LIN {X 0,Y 185.701,Z 460.549,A -85,B 0,C 180,E1 -22371.274,E2 -22371.274} C_VEL
LIN {X 0,Y 187.738,Z 470.881,A -85,B 0,C 180,E1 -22375.839,E2 -22375.839} C_VEL
LIN {X 0,Y 188.686,Z 475.361,A -85,B 0,C 180,E1 -22377.768,E2 -22377.768} C_VEL
LIN {X 0,Y 191.548,Z 486.797,A -85,B 0,C 180,E1 -22378.685,E2 -22378.685} C_VEL
LIN {X 0,Y 193.659,Z 519.979,A -85,B 0,C 180,E1 -22380.8,E2 -22380.8} C_VEL
LIN {X 0,Y 195.142,Z 539.248,A -85,B 0,C 180,E1 -22382.01,E2 -22382.01} C_VEL
LIN {X 0,Y 192.666,Z 586.047,A -85,B 0,C 180,E1 -22384.693,E2 -22384.693} C_VEL
LIN {X 0,Y 191.547,Z 599.858,A -85,B 0,C 180,E1 -22385.91,E2 -22385.91} C_VEL
LIN {X 0,Y 190.024,Z 613.54,A -85,B 0,C 180,E1 -22387.612,E2 -22387.612} C_VEL
LIN {X 0,Y 188.629,Z 625.455,A -85,B 0,C 180,E1 -22389.556,E2 -22389.556} C_VEL
LIN {X 0,Y 188.498,Z 626.394,A -85,B 0,C 180,E1 -22389.737,E2 -22389.737} C_VEL
LIN {X 0,Y 187.176,Z 631.288,A -85,B 0,C 180,E1 -22390.708,E2 -22390.708} C_VEL
LIN {X 0,Y 183.337,Z 638.645,A -85,B 0,C 180,E1 -22392.419,E2 -22392.419} C_VEL
LIN {X 0,Y 179.646,Z 645.469,A -85,B 0,C 180,E1 -22394.364,E2 -22394.364} C_VEL
LIN {X 0,Y 178.558,Z 649.547,A -85,B 0,C 180,E1 -22395.664,E2 -22395.664} C_VEL
LIN {X 0,Y 177.85,Z 657.711,A -85,B 0,C 180,E1 -22398.605,E2 -22398.605} C_VEL
LIN {X 0,Y 177.522,Z 664.858,A -85,B 0,C 180,E1 -22401.787,E2 -22401.787} C_VEL
LIN {X 0,Y 177.494,Z 671.375,A -85,B 0,C 180,E1 -22405.459,E2 -22405.459} C_VEL
LIN {X 0,Y 177.626,Z 675.992,A -85,B 0,C 180,E1 -22408.867,E2 -22408.867} C_VEL
LIN {X 0,Y 177.383,Z 678.317,A -85,B 0,C 180,E1 -22411.136,E2 -22411.136} C_VEL
LIN {X 0,Y 176.849,Z 680.76,A -85,B 0,C 180,E1 -22414.56,E2 -22414.56} C_VEL
LIN {X 0,Y 176.648,Z 681.882,A -85,B 0,C 180,E1 -22416.856,E2 -22416.856} C_VEL
LIN {X 0,Y 176.961,Z 682.934,A -85,B 0,C 180,E1 -22421.455,E2 -22421.455} C_VEL
LIN {X 0,Y 178.495,Z 682.536,A -85,B 0,C 180,E1 -22426,E2 -22426} C_VEL
LIN {X 0,Y 181.429,Z 680.73,A -85,B 0,C 180,E1 -22430.405,E2 -22430.405} C_VEL
LIN {X 0,Y 185.547,Z 677.444,A -85,B 0,C 180,E1 -22434.624,E2 -22434.624} C_VEL
LIN {X 0,Y 189.455,Z 673.992,A -85,B 0,C 180,E1 -22437.627,E2 -22437.627} C_VEL
LIN {X 0,Y 195.633,Z 667.93,A -85,B 0,C 180,E1 -22441.394,E2 -22441.394} C_VEL
LIN {X 0,Y 202.062,Z 661.103,A -85,B 0,C 180,E1 -22444.417,E2 -22444.417} C_VEL
LIN {X 0,Y 209.177,Z 652.611,A -85,B 0,C 180,E1 -22447.213,E2 -22447.213} C_VEL
LIN {X 0,Y 215.799,Z 643.753,A -85,B 0,C 180,E1 -22449.426,E2 -22449.426} C_VEL
LIN {X 0,Y 222.976,Z 632.961,A -85,B 0,C 180,E1 -22451.446,E2 -22451.446} C_VEL
LIN {X 0,Y 229.411,Z 621.99,A -85,B 0,C 180,E1 -22452.972,E2 -22452.972} C_VEL
LIN {X 0,Y 235.662,Z 609.39,A -85,B 0,C 180,E1 -22454.31,E2 -22454.31} C_VEL
LIN {X 0,Y 240.513,Z 597.54,A -85,B 0,C 180,E1 -22455.274,E2 -22455.274} C_VEL
LIN {X 0,Y 244.965,Z 584.543,A -85,B 0,C 180,E1 -22456.036,E2 -22456.036} C_VEL
LIN {X 0,Y 248.669,Z 569.68,A -85,B 0,C 180,E1 -22456.721,E2 -22456.721} C_VEL
LIN {X 0,Y 251.184,Z 556.435,A -85,B 0,C 180,E1 -22457.281,E2 -22457.281} C_VEL
LIN {X 0,Y 250.72,Z 552.705,A -85,B 0,C 180,E1 -22459.004,E2 -22459.004} C_VEL
LIN {X 0,Y 250.494,Z 550.56,A -85,B 0,C 180,E1 -22460.257,E2 -22460.257} C_VEL
LIN {X 0,Y 250.39,Z 547.96,A -85,B 0,C 180,E1 -22462.942,E2 -22462.942} C_VEL
LIN {X 0,Y 250.635,Z 547.364,A -85,B 0,C 180,E1 -22464.409,E2 -22464.409} C_VEL
LIN {X 0,Y 251.66,Z 547.678,A -85,B 0,C 180,E1 -22467.346,E2 -22467.346} C_VEL
LIN {X 0,Y 252.275,Z 548.822,A -85,B 0,C 180,E1 -22468.664,E2 -22468.664} C_VEL
LIN {X 0,Y 248.421,Z 568.129,A -85,B 0,C 180,E1 -22469.52,E2 -22469.52} C_VEL
LIN {X 0,Y 244.81,Z 581.444,A -85,B 0,C 180,E1 -22470.419,E2 -22470.419} C_VEL
LIN {X 0,Y 240.18,Z 594.192,A -85,B 0,C 180,E1 -22471.554,E2 -22471.554} C_VEL
LIN {X 0,Y 235.167,Z 605.631,A -85,B 0,C 180,E1 -22472.887,E2 -22472.887} C_VEL
LIN {X 0,Y 229.144,Z 616.854,A -85,B 0,C 180,E1 -22474.571,E2 -22474.571} C_VEL
LIN {X 0,Y 223.649,Z 625.549,A -85,B 0,C 180,E1 -22476.239,E2 -22476.239} C_VEL
LIN {X 0,Y 217.842,Z 633.74,A -85,B 0,C 180,E1 -22478.222,E2 -22478.222} C_VEL
LIN {X 0,Y 211.559,Z 641.305,A -85,B 0,C 180,E1 -22480.597,E2 -22480.597} C_VEL
LIN {X 0,Y 205.668,Z 647.446,A -85,B 0,C 180,E1 -22483.101,E2 -22483.101} C_VEL
LIN {X 0,Y 200.307,Z 652.348,A -85,B 0,C 180,E1 -22485.782,E2 -22485.782} C_VEL
LIN {X 0,Y 195.383,Z 656.121,A -85,B 0,C 180,E1 -22488.589,E2 -22488.589} C_VEL
LIN {X 0,Y 191.066,Z 658.891,A -85,B 0,C 180,E1 -22491.539,E2 -22491.539} C_VEL
LIN {X 0,Y 188.458,Z 660.203,A -85,B 0,C 180,E1 -22493.576,E2 -22493.576} C_VEL
LIN {X 0,Y 186.12,Z 661.109,A -85,B 0,C 180,E1 -22495.669,E2 -22495.669} C_VEL
LIN {X 0,Y 182.445,Z 661.688,A -85,B 0,C 180,E1 -22499.684,E2 -22499.684} C_VEL
LIN {X 0,Y 180.64,Z 661.354,A -85,B 0,C 180,E1 -22502.23,E2 -22502.23} C_VEL
LIN {X 0,Y 179.301,Z 660.645,A -85,B 0,C 180,E1 -22504.496,E2 -22504.496} C_VEL
LIN {X 0,Y 177.655,Z 658.413,A -85,B 0,C 180,E1 -22508.502,E2 -22508.502} C_VEL
LIN {X 0,Y 176.659,Z 654.746,A -85,B 0,C 180,E1 -22512.639,E2 -22512.639} C_VEL
LIN {X 0,Y 176.419,Z 650.464,A -85,B 0,C 180,E1 -22516.192,E2 -22516.192} C_VEL
LIN {X 0,Y 176.624,Z 643.895,A -85,B 0,C 180,E1 -22520.375,E2 -22520.375} C_VEL
LIN {X 0,Y 177.27,Z 636.508,A -85,B 0,C 180,E1 -22524.01,E2 -22524.01} C_VEL
LIN {X 0,Y 178.251,Z 627.333,A -85,B 0,C 180,E1 -22527.599,E2 -22527.599} C_VEL
LIN {X 0,Y 179.439,Z 617.727,A -85,B 0,C 180,E1 -22530.608,E2 -22530.608} C_VEL
LIN {X 0,Y 180.967,Z 605.843,A -85,B 0,C 180,E1 -22533.601,E2 -22533.601} C_VEL
LIN {X 0,Y 182.418,Z 593.758,A -85,B 0,C 180,E1 -22535.994,E2 -22535.994} C_VEL
LIN {X 0,Y 183.934,Z 580.594,A -85,B 0,C 180,E1 -22538.034,E2 -22538.034} C_VEL
LIN {X 0,Y 185.179,Z 566.664,A -85,B 0,C 180,E1 -22539.648,E2 -22539.648} C_VEL
LIN {X 0,Y 186.107,Z 553.364,A -85,B 0,C 180,E1 -22540.742,E2 -22540.742} C_VEL
LIN {X 0,Y 189.303,Z 493.801,A -85,B 0,C 180,E1 -22544.168,E2 -22544.168} C_VEL
LIN {X 0,Y 178.456,Z 461.253,A -85,B 0,C 180,E1 -22547.11,E2 -22547.11} C_VEL
LIN {X 0,Y 178.409,Z 461.26,A -85,B 0,C 180,E1 -22551.985,E2 -22551.985} C_VEL
LIN {X 0,Y 178.485,Z 461.252,A -85,B 0,C 180,E1 -22556.545,E2 -22556.545} C_VEL
LIN {X 0,Y 178.445,Z 461.254,A -85,B 0,C 180,E1 -22561.795,E2 -22561.795} C_VEL
LIN {X 0,Y 178.517,Z 461.247,A -85,B 0,C 180,E1 -22564.888,E2 -22564.888} C_VEL
LIN {X 0,Y 178.624,Z 461.23,A -85,B 0,C 180,E1 -22570.784,E2 -22570.784} C_VEL
LIN {X 0,Y 178.659,Z 461.232,A -85,B 0,C 180,E1 -22576.347,E2 -22576.347} C_VEL
LIN {X 0,Y 178.906,Z 461.196,A -85,B 0,C 180,E1 -22580.959,E2 -22580.959} C_VEL
LIN {X 0,Y 179.148,Z 461.166,A -85,B 0,C 180,E1 -22587.751,E2 -22587.751} C_VEL
LIN {X 0,Y 179.364,Z 461.138,A -85,B 0,C 180,E1 -22589.999,E2 -22589.999} C_VEL
LIN {X 0,Y 178.857,Z 461.206,A -85,B 0,C 180,E1 -22594.507,E2 -22594.507} C_VEL
LIN {X 0,Y 178.911,Z 461.196,A -85,B 0,C 180,E1 -22599.039,E2 -22599.039} C_VEL
LIN {X 0,Y 178.652,Z 461.229,A -85,B 0,C 180,E1 -22603.652,E2 -22603.652} C_VEL
LIN {X 0,Y 178.62,Z 461.234,A -85,B 0,C 180,E1 -22609.212,E2 -22609.212} C_VEL
LIN {X 0,Y 178.515,Z 461.243,A -85,B 0,C 180,E1 -22615.11,E2 -22615.11} C_VEL
LIN {X 0,Y 178.459,Z 461.255,A -85,B 0,C 180,E1 -22620.794,E2 -22620.794} C_VEL
LIN {X 0,Y 178.482,Z 461.248,A -85,B 0,C 180,E1 -22624.218,E2 -22624.218} C_VEL
LIN {X 0,Y 178.388,Z 461.263,A -85,B 0,C 180,E1 -22629.075,E2 -22629.075} C_VEL
LIN {X 0,Y 178.393,Z 461.26,A -85,B 0,C 180,E1 -22632.046,E2 -22632.046} C_VEL
LIN {X 0,Y 178.391,Z 461.262,A -85,B 0,C 180,E1 -22635.164,E2 -22635.164} C_VEL
LIN {X 0,Y 178.401,Z 461.263,A -85,B 0,C 180,E1 -22638.459,E2 -22638.459} C_VEL
LIN {X 0,Y 178.421,Z 461.257,A -85,B 0,C 180,E1 -22643.783,E2 -22643.783} C_VEL
LIN {X 0,Y 178.484,Z 461.254,A -85,B 0,C 180,E1 -22646.546,E2 -22646.546} C_VEL
LIN {X 0,Y 178.52,Z 461.243,A -85,B 0,C 180,E1 -22650.007,E2 -22650.007} C_VEL
LIN {X 0,Y 178.533,Z 461.246,A -85,B 0,C 180,E1 -22654.876,E2 -22654.876} C_VEL
LIN {X 0,Y 178.638,Z 461.232,A -85,B 0,C 180,E1 -22660.769,E2 -22660.769} C_VEL
LIN {X 0,Y 178.671,Z 461.228,A -85,B 0,C 180,E1 -22664.018,E2 -22664.018} C_VEL
LIN {X 0,Y 178.857,Z 461.203,A -85,B 0,C 180,E1 -22669.214,E2 -22669.214} C_VEL
LIN {X 0,Y 178.926,Z 461.195,A -85,B 0,C 180,E1 -22673.233,E2 -22673.233} C_VEL
LIN {X 0,Y 179.152,Z 461.165,A -85,B 0,C 180,E1 -22677.752,E2 -22677.752} C_VEL
LIN {X 0,Y 179.369,Z 461.141,A -85,B 0,C 180,E1 -22680,E2 -22680} C_VEL
LIN {X 0,Y 178.874,Z 461.2,A -85,B 0,C 180,E1 -22684.507,E2 -22684.507} C_VEL
LIN {X 0,Y 178.974,Z 461.191,A -85,B 0,C 180,E1 -22689.037,E2 -22689.037} C_VEL
LIN {X 0,Y 178.681,Z 461.221,A -85,B 0,C 180,E1 -22693.651,E2 -22693.651} C_VEL
LIN {X 0,Y 178.621,Z 461.234,A -85,B 0,C 180,E1 -22699.216,E2 -22699.216} C_VEL
LIN {X 0,Y 178.519,Z 461.247,A -85,B 0,C 180,E1 -22705.115,E2 -22705.115} C_VEL
LIN {X 0,Y 178.501,Z 461.246,A -85,B 0,C 180,E1 -22710.787,E2 -22710.787} C_VEL
LIN {X 0,Y 178.485,Z 461.251,A -85,B 0,C 180,E1 -22714.22,E2 -22714.22} C_VEL
LIN {X 0,Y 178.395,Z 461.258,A -85,B 0,C 180,E1 -22719.075,E2 -22719.075} C_VEL
LIN {X 0,Y 178.398,Z 461.26,A -85,B 0,C 180,E1 -22722.045,E2 -22722.045} C_VEL
LIN {X 0,Y 178.394,Z 461.263,A -85,B 0,C 180,E1 -22725.164,E2 -22725.164} C_VEL
LIN {X 0,Y 178.599,Z 461.379,A -85,B 0,C 180,E1 -22730.979,E2 -22730.979} C_VEL
LIN {X 0,Y 180.643,Z 471.556,A -85,B 0,C 180,E1 -22735.659,E2 -22735.659} C_VEL
LIN {X 0,Y 181.369,Z 475.028,A -85,B 0,C 180,E1 -22737.147,E2 -22737.147} C_VEL
LIN {X 0,Y 184.69,Z 487.892,A -85,B 0,C 180,E1 -22738.233,E2 -22738.233} C_VEL
LIN {X 0,Y 186.699,Z 520.317,A -85,B 0,C 180,E1 -22740.381,E2 -22740.381} C_VEL
LIN {X 0,Y 188.159,Z 539.471,A -85,B 0,C 180,E1 -22741.637,E2 -22741.637} C_VEL
LIN {X 0,Y 185.629,Z 585.844,A -85,B 0,C 180,E1 -22744.416,E2 -22744.416} C_VEL
LIN {X 0,Y 184.49,Z 599.914,A -85,B 0,C 180,E1 -22745.722,E2 -22745.722} C_VEL
LIN {X 0,Y 182.927,Z 613.572,A -85,B 0,C 180,E1 -22747.508,E2 -22747.508} C_VEL
LIN {X 0,Y 181.442,Z 625.783,A -85,B 0,C 180,E1 -22749.616,E2 -22749.616} C_VEL
LIN {X 0,Y 180.084,Z 637.05,A -85,B 0,C 180,E1 -22752.102,E2 -22752.102} C_VEL
LIN {X 0,Y 178.904,Z 646.257,A -85,B 0,C 180,E1 -22754.624,E2 -22754.624} C_VEL
LIN {X 0,Y 178.558,Z 649.547,A -85,B 0,C 180,E1 -22755.664,E2 -22755.664} C_VEL
LIN {X 0,Y 177.546,Z 653.521,A -85,B 0,C 180,E1 -22757.032,E2 -22757.032} C_VEL
LIN {X 0,Y 174.285,Z 659.229,A -85,B 0,C 180,E1 -22759.452,E2 -22759.452} C_VEL
LIN {X 0,Y 171.212,Z 664.277,A -85,B 0,C 180,E1 -22762.125,E2 -22762.125} C_VEL
LIN {X 0,Y 170.513,Z 667.229,A -85,B 0,C 180,E1 -22763.845,E2 -22763.845} C_VEL
LIN {X 0,Y 170.596,Z 672.954,A -85,B 0,C 180,E1 -22767.64,E2 -22767.64} C_VEL
LIN {X 0,Y 170.668,Z 675.747,A -85,B 0,C 180,E1 -22770.001,E2 -22770.001} C_VEL
LIN {X 0,Y 170.245,Z 677.883,A -85,B 0,C 180,E1 -22772.367,E2 -22772.367} C_VEL
LIN {X 0,Y 169.72,Z 680.438,A -85,B 0,C 180,E1 -22776.368,E2 -22776.368} C_VEL
LIN {X 0,Y 169.645,Z 681.621,A -85,B 0,C 180,E1 -22779.539,E2 -22779.539} C_VEL
LIN {X 0,Y 170.666,Z 682.248,A -85,B 0,C 180,E1 -22784.306,E2 -22784.306} C_VEL
LIN {X 0,Y 173.115,Z 681.425,A -85,B 0,C 180,E1 -22788.953,E2 -22788.953} C_VEL
LIN {X 0,Y 176.794,Z 679.2,A -85,B 0,C 180,E1 -22793.425,E2 -22793.425} C_VEL
LIN {X 0,Y 181.757,Z 675.549,A -85,B 0,C 180,E1 -22797.647,E2 -22797.647} C_VEL
LIN {X 0,Y 186.362,Z 671.786,A -85,B 0,C 180,E1 -22800.605,E2 -22800.605} C_VEL
LIN {X 0,Y 191.512,Z 667.071,A -85,B 0,C 180,E1 -22803.4,E2 -22803.4} C_VEL
LIN {X 0,Y 198.38,Z 660.316,A -85,B 0,C 180,E1 -22806.4,E2 -22806.4} C_VEL
LIN {X 0,Y 204.815,Z 653.196,A -85,B 0,C 180,E1 -22808.773,E2 -22808.773} C_VEL
LIN {X 0,Y 211.719,Z 644.664,A -85,B 0,C 180,E1 -22810.966,E2 -22810.966} C_VEL
LIN {X 0,Y 219.17,Z 634.332,A -85,B 0,C 180,E1 -22812.955,E2 -22812.955} C_VEL
LIN {X 0,Y 225.823,Z 623.791,A -85,B 0,C 180,E1 -22814.447,E2 -22814.447} C_VEL
LIN {X 0,Y 231.994,Z 612.482,A -85,B 0,C 180,E1 -22815.7,E2 -22815.7} C_VEL
LIN {X 0,Y 237.79,Z 599.752,A -85,B 0,C 180,E1 -22816.782,E2 -22816.782} C_VEL
LIN {X 0,Y 242.47,Z 587.137,A -85,B 0,C 180,E1 -22817.529,E2 -22817.529} C_VEL
LIN {X 0,Y 246.909,Z 571.217,A -85,B 0,C 180,E1 -22818.276,E2 -22818.276} C_VEL
LIN {X 0,Y 249.076,Z 560.769,A -85,B 0,C 180,E1 -22818.712,E2 -22818.712} C_VEL
LIN {X 0,Y 248.802,Z 557.233,A -85,B 0,C 180,E1 -22820.64,E2 -22820.64} C_VEL
LIN {X 0,Y 248.861,Z 554.658,A -85,B 0,C 180,E1 -22823.383,E2 -22823.383} C_VEL
LIN {X 0,Y 249.34,Z 554.291,A -85,B 0,C 180,E1 -22825.686,E2 -22825.686} C_VEL
LIN {X 0,Y 250.017,Z 554.637,A -85,B 0,C 180,E1 -22827.235,E2 -22827.235} C_VEL
LIN {X 0,Y 246.333,Z 571.491,A -85,B 0,C 180,E1 -22828.075,E2 -22828.075} C_VEL
LIN {X 0,Y 242.221,Z 584.894,A -85,B 0,C 180,E1 -22829.001,E2 -22829.001} C_VEL
LIN {X 0,Y 237.736,Z 596.488,A -85,B 0,C 180,E1 -22830.057,E2 -22830.057} C_VEL
LIN {X 0,Y 232.572,Z 607.309,A -85,B 0,C 180,E1 -22831.319,E2 -22831.319} C_VEL
LIN {X 0,Y 225.615,Z 619.36,A -85,B 0,C 180,E1 -22833.148,E2 -22833.148} C_VEL
LIN {X 0,Y 219.543,Z 628.275,A -85,B 0,C 180,E1 -22834.902,E2 -22834.902} C_VEL
LIN {X 0,Y 212.619,Z 636.953,A -85,B 0,C 180,E1 -22837.145,E2 -22837.145} C_VEL
LIN {X 0,Y 206.117,Z 644.087,A -85,B 0,C 180,E1 -22839.543,E2 -22839.543} C_VEL
LIN {X 0,Y 200.931,Z 648.956,A -85,B 0,C 180,E1 -22841.651,E2 -22841.651} C_VEL
LIN {X 0,Y 195.276,Z 653.63,A -85,B 0,C 180,E1 -22844.34,E2 -22844.34} C_VEL
LIN {X 0,Y 190.04,Z 657.289,A -85,B 0,C 180,E1 -22847.18,E2 -22847.18} C_VEL
LIN {X 0,Y 185.499,Z 659.837,A -85,B 0,C 180,E1 -22850.09,E2 -22850.09} C_VEL
LIN {X 0,Y 181.3,Z 661.572,A -85,B 0,C 180,E1 -22853.322,E2 -22853.322} C_VEL
LIN {X 0,Y 176.771,Z 662.426,A -85,B 0,C 180,E1 -22857.721,E2 -22857.721} C_VEL
LIN {X 0,Y 174.956,Z 662.226,A -85,B 0,C 180,E1 -22860,E2 -22860} C_VEL
LIN {X 0,Y 172.03,Z 660.637,A -85,B 0,C 180,E1 -22864.687,E2 -22864.687} C_VEL
LIN {X 0,Y 170.54,Z 658.221,A -85,B 0,C 180,E1 -22868.481,E2 -22868.481} C_VEL
LIN {X 0,Y 169.664,Z 655.105,A -85,B 0,C 180,E1 -22871.953,E2 -22871.953} C_VEL
LIN {X 0,Y 169.34,Z 650.753,A -85,B 0,C 180,E1 -22875.65,E2 -22875.65} C_VEL
LIN {X 0,Y 169.442,Z 645.131,A -85,B 0,C 180,E1 -22879.379,E2 -22879.379} C_VEL
LIN {X 0,Y 169.988,Z 638.049,A -85,B 0,C 180,E1 -22883.127,E2 -22883.127} C_VEL
LIN {X 0,Y 170.962,Z 629.103,A -85,B 0,C 180,E1 -22886.884,E2 -22886.884} C_VEL
LIN {X 0,Y 172.01,Z 620.202,A -85,B 0,C 180,E1 -22889.922,E2 -22889.922} C_VEL
LIN {X 0,Y 173.341,Z 609.586,A -85,B 0,C 180,E1 -22892.839,E2 -22892.839} C_VEL
LIN {X 0,Y 174.77,Z 598.414,A -85,B 0,C 180,E1 -22895.314,E2 -22895.314} C_VEL
LIN {X 0,Y 176.285,Z 586.092,A -85,B 0,C 180,E1 -22897.484,E2 -22897.484} C_VEL
LIN {X 0,Y 177.597,Z 572.798,A -85,B 0,C 180,E1 -22899.284,E2 -22899.284} C_VEL
LIN {X 0,Y 178.742,Z 559.118,A -85,B 0,C 180,E1 -22900.634,E2 -22900.634} C_VEL
LIN {X 0,Y 179.933,Z 536.769,A -85,B 0,C 180,E1 -22902.096,E2 -22902.096} C_VEL
LIN {X 0,Y 182.328,Z 494.869,A -85,B 0,C 180,E1 -22904.608,E2 -22904.608} C_VEL
LIN {X 0,Y 171.384,Z 462.134,A -85,B 0,C 180,E1 -22907.705,E2 -22907.705} C_VEL
LIN {X 0,Y 171.361,Z 462.139,A -85,B 0,C 180,E1 -22912.033,E2 -22912.033} C_VEL
LIN {X 0,Y 171.399,Z 462.131,A -85,B 0,C 180,E1 -22915.092,E2 -22915.092} C_VEL
LIN {X 0,Y 171.41,Z 462.132,A -85,B 0,C 180,E1 -22920.526,E2 -22920.526} C_VEL
LIN {X 0,Y 171.444,Z 462.127,A -85,B 0,C 180,E1 -22925.799,E2 -22925.799} C_VEL
LIN {X 0,Y 171.58,Z 462.106,A -85,B 0,C 180,E1 -22930.871,E2 -22930.871} C_VEL
LIN {X 0,Y 171.577,Z 462.112,A -85,B 0,C 180,E1 -22935.772,E2 -22935.772} C_VEL
LIN {X 0,Y 171.844,Z 462.075,A -85,B 0,C 180,E1 -22940.584,E2 -22940.584} C_VEL
LIN {X 0,Y 171.804,Z 462.083,A -85,B 0,C 180,E1 -22945.306,E2 -22945.306} C_VEL
LIN {X 0,Y 172.328,Z 462.014,A -85,B 0,C 180,E1 -22949.999,E2 -22949.999} C_VEL
LIN {X 0,Y 171.806,Z 462.083,A -85,B 0,C 180,E1 -22954.692,E2 -22954.692} C_VEL
LIN {X 0,Y 171.848,Z 462.075,A -85,B 0,C 180,E1 -22959.414,E2 -22959.414} C_VEL
LIN {X 0,Y 171.569,Z 462.113,A -85,B 0,C 180,E1 -22964.227,E2 -22964.227} C_VEL
LIN {X 0,Y 171.539,Z 462.115,A -85,B 0,C 180,E1 -22969.555,E2 -22969.555} C_VEL
LIN {X 0,Y 171.443,Z 462.123,A -85,B 0,C 180,E1 -22975.598,E2 -22975.598} C_VEL
LIN {X 0,Y 171.417,Z 462.133,A -85,B 0,C 180,E1 -22980.572,E2 -22980.572} C_VEL
LIN {X 0,Y 171.391,Z 462.133,A -85,B 0,C 180,E1 -22985.034,E2 -22985.034} C_VEL
LIN {X 0,Y 171.343,Z 462.142,A -85,B 0,C 180,E1 -22988.801,E2 -22988.801} C_VEL
LIN {X 0,Y 171.318,Z 462.141,A -85,B 0,C 180,E1 -22994.217,E2 -22994.217} C_VEL
LIN {X 0,Y 171.334,Z 462.141,A -85,B 0,C 180,E1 -22998.981,E2 -22998.981} C_VEL
LIN {X 0,Y 171.385,Z 462.13,A -85,B 0,C 180,E1 -23002.041,E2 -23002.041} C_VEL
LIN {X 0,Y 171.397,Z 462.135,A -85,B 0,C 180,E1 -23005.092,E2 -23005.092} C_VEL
LIN {X 0,Y 171.447,Z 462.124,A -85,B 0,C 180,E1 -23010.534,E2 -23010.534} C_VEL
LIN {X 0,Y 171.458,Z 462.126,A -85,B 0,C 180,E1 -23015.802,E2 -23015.802} C_VEL
LIN {X 0,Y 171.594,Z 462.11,A -85,B 0,C 180,E1 -23020.874,E2 -23020.874} C_VEL
LIN {X 0,Y 171.596,Z 462.107,A -85,B 0,C 180,E1 -23025.775,E2 -23025.775} C_VEL
LIN {X 0,Y 171.889,Z 462.074,A -85,B 0,C 180,E1 -23030.587,E2 -23030.587} C_VEL
LIN {X 0,Y 171.82,Z 462.077,A -85,B 0,C 180,E1 -23035.308,E2 -23035.308} C_VEL
LIN {X 0,Y 172.332,Z 462.017,A -85,B 0,C 180,E1 -23040,E2 -23040} C_VEL
LIN {X 0,Y 171.823,Z 462.078,A -85,B 0,C 180,E1 -23044.693,E2 -23044.693} C_VEL
LIN {X 0,Y 171.907,Z 462.07,A -85,B 0,C 180,E1 -23049.412,E2 -23049.412} C_VEL
LIN {X 0,Y 171.594,Z 462.105,A -85,B 0,C 180,E1 -23054.226,E2 -23054.226} C_VEL
LIN {X 0,Y 171.541,Z 462.115,A -85,B 0,C 180,E1 -23059.56,E2 -23059.56} C_VEL
LIN {X 0,Y 171.458,Z 462.126,A -85,B 0,C 180,E1 -23065.61,E2 -23065.61} C_VEL
LIN {X 0,Y 171.458,Z 462.124,A -85,B 0,C 180,E1 -23070.597,E2 -23070.597} C_VEL
LIN {X 0,Y 171.392,Z 462.136,A -85,B 0,C 180,E1 -23075.035,E2 -23075.035} C_VEL
LIN {X 0,Y 171.357,Z 462.136,A -85,B 0,C 180,E1 -23078.808,E2 -23078.808} C_VEL
LIN {X 0,Y 171.321,Z 462.144,A -85,B 0,C 180,E1 -23084.218,E2 -23084.218} C_VEL
LIN {X 0,Y 171.502,Z 462.119,A -85,B 0,C 180,E1 -23090.579,E2 -23090.579} C_VEL
LIN {X 0,Y 173.542,Z 472.168,A -85,B 0,C 180,E1 -23095.462,E2 -23095.462} C_VEL
LIN {X 0,Y 173.972,Z 474.305,A -85,B 0,C 180,E1 -23096.459,E2 -23096.459} C_VEL
LIN {X 0,Y 177.844,Z 489.066,A -85,B 0,C 180,E1 -23097.756,E2 -23097.756} C_VEL
LIN {X 0,Y 179.756,Z 520.758,A -85,B 0,C 180,E1 -23099.937,E2 -23099.937} C_VEL
LIN {X 0,Y 181.179,Z 540.044,A -85,B 0,C 180,E1 -23101.264,E2 -23101.264} C_VEL
LIN {X 0,Y 178.679,Z 584.578,A -85,B 0,C 180,E1 -23104.051,E2 -23104.051} C_VEL
LIN {X 0,Y 177.556,Z 598.633,A -85,B 0,C 180,E1 -23105.396,E2 -23105.396} C_VEL
LIN {X 0,Y 175.989,Z 611.81,A -85,B 0,C 180,E1 -23107.165,E2 -23107.165} C_VEL
LIN {X 0,Y 174.49,Z 624.286,A -85,B 0,C 180,E1 -23109.365,E2 -23109.365} C_VEL
LIN {X 0,Y 173.118,Z 635.756,A -85,B 0,C 180,E1 -23111.969,E2 -23111.969} C_VEL
LIN {X 0,Y 171.904,Z 645.068,A -85,B 0,C 180,E1 -23114.59,E2 -23114.59} C_VEL
LIN {X 0,Y 171.148,Z 653.703,A -85,B 0,C 180,E1 -23117.551,E2 -23117.551} C_VEL
LIN {X 0,Y 170.577,Z 661.794,A -85,B 0,C 180,E1 -23121.012,E2 -23121.012} C_VEL
LIN {X 0,Y 170.513,Z 667.229,A -85,B 0,C 180,E1 -23123.845,E2 -23123.845} C_VEL
LIN {X 0,Y 169.84,Z 669.942,A -85,B 0,C 180,E1 -23125.605,E2 -23125.605} C_VEL
LIN {X 0,Y 168.256,Z 672.115,A -85,B 0,C 180,E1 -23127.404,E2 -23127.404} C_VEL
LIN {X 0,Y 164.424,Z 675.542,A -85,B 0,C 180,E1 -23131.183,E2 -23131.183} C_VEL
LIN {X 0,Y 163.025,Z 677.475,A -85,B 0,C 180,E1 -23133.88,E2 -23133.88} C_VEL
LIN {X 0,Y 162.658,Z 679.622,A -85,B 0,C 180,E1 -23137.449,E2 -23137.449} C_VEL
LIN {X 0,Y 163.067,Z 681.206,A -85,B 0,C 180,E1 -23142.445,E2 -23142.445} C_VEL
LIN {X 0,Y 164.867,Z 681.393,A -85,B 0,C 180,E1 -23147.362,E2 -23147.362} C_VEL
LIN {X 0,Y 168.164,Z 680.215,A -85,B 0,C 180,E1 -23152.095,E2 -23152.095} C_VEL
LIN {X 0,Y 172.733,Z 677.628,A -85,B 0,C 180,E1 -23156.588,E2 -23156.588} C_VEL
LIN {X 0,Y 178.616,Z 673.581,A -85,B 0,C 180,E1 -23160.765,E2 -23160.765} C_VEL
LIN {X 0,Y 185.676,Z 668.028,A -85,B 0,C 180,E1 -23164.596,E2 -23164.596} C_VEL
LIN {X 0,Y 192.807,Z 661.677,A -85,B 0,C 180,E1 -23167.631,E2 -23167.631} C_VEL
LIN {X 0,Y 200.613,Z 653.822,A -85,B 0,C 180,E1 -23170.4,E2 -23170.4} C_VEL
LIN {X 0,Y 207.8,Z 645.644,A -85,B 0,C 180,E1 -23172.566,E2 -23172.566} C_VEL
LIN {X 0,Y 215.529,Z 635.756,A -85,B 0,C 180,E1 -23174.514,E2 -23174.514} C_VEL
LIN {X 0,Y 221.831,Z 626.654,A -85,B 0,C 180,E1 -23175.858,E2 -23175.858} C_VEL
LIN {X 0,Y 228.713,Z 615.037,A -85,B 0,C 180,E1 -23177.193,E2 -23177.193} C_VEL
LIN {X 0,Y 235.227,Z 601.98,A -85,B 0,C 180,E1 -23178.327,E2 -23178.327} C_VEL
LIN {X 0,Y 240.808,Z 588.272,A -85,B 0,C 180,E1 -23179.137,E2 -23179.137} C_VEL
LIN {X 0,Y 245.118,Z 574.249,A -85,B 0,C 180,E1 -23179.793,E2 -23179.793} C_VEL
LIN {X 0,Y 247.164,Z 565.427,A -85,B 0,C 180,E1 -23180.196,E2 -23180.196} C_VEL
LIN {X 0,Y 247.177,Z 563.443,A -85,B 0,C 180,E1 -23181.454,E2 -23181.454} C_VEL
LIN {X 0,Y 247.349,Z 561.484,A -85,B 0,C 180,E1 -23183.677,E2 -23183.677} C_VEL
LIN {X 0,Y 247.841,Z 561.257,A -85,B 0,C 180,E1 -23185.916,E2 -23185.916} C_VEL
LIN {X 0,Y 245.069,Z 572.959,A -85,B 0,C 180,E1 -23186.487,E2 -23186.487} C_VEL
LIN {X 0,Y 240.86,Z 585.994,A -85,B 0,C 180,E1 -23187.366,E2 -23187.366} C_VEL
LIN {X 0,Y 236.172,Z 597.354,A -85,B 0,C 180,E1 -23188.366,E2 -23188.366} C_VEL
LIN {X 0,Y 229.451,Z 610.476,A -85,B 0,C 180,E1 -23189.911,E2 -23189.911} C_VEL
LIN {X 0,Y 222.995,Z 620.916,A -85,B 0,C 180,E1 -23191.505,E2 -23191.505} C_VEL
LIN {X 0,Y 215.897,Z 630.475,A -85,B 0,C 180,E1 -23193.41,E2 -23193.41} C_VEL
LIN {X 0,Y 209.725,Z 637.799,A -85,B 0,C 180,E1 -23195.3,E2 -23195.3} C_VEL
LIN {X 0,Y 202.938,Z 644.733,A -85,B 0,C 180,E1 -23197.608,E2 -23197.608} C_VEL
LIN {X 0,Y 196.367,Z 650.493,A -85,B 0,C 180,E1 -23200.122,E2 -23200.122} C_VEL
LIN {X 0,Y 190.387,Z 655.006,A -85,B 0,C 180,E1 -23202.823,E2 -23202.823} C_VEL
LIN {X 0,Y 183.084,Z 659.375,A -85,B 0,C 180,E1 -23206.684,E2 -23206.684} C_VEL
LIN {X 0,Y 178.664,Z 661.412,A -85,B 0,C 180,E1 -23209.555,E2 -23209.555} C_VEL
LIN {X 0,Y 174.137,Z 662.773,A -85,B 0,C 180,E1 -23213.046,E2 -23213.046} C_VEL
LIN {X 0,Y 169.515,Z 663.047,A -85,B 0,C 180,E1 -23217.624,E2 -23217.624} C_VEL
LIN {X 0,Y 167.69,Z 662.597,A -85,B 0,C 180,E1 -23220,E2 -23220} C_VEL
LIN {X 0,Y 164.745,Z 660.451,A -85,B 0,C 180,E1 -23224.894,E2 -23224.894} C_VEL
LIN {X 0,Y 163.428,Z 657.93,A -85,B 0,C 180,E1 -23228.466,E2 -23228.466} C_VEL
LIN {X 0,Y 162.503,Z 654.056,A -85,B 0,C 180,E1 -23232.488,E2 -23232.488} C_VEL
LIN {X 0,Y 162.235,Z 649.229,A -85,B 0,C 180,E1 -23236.354,E2 -23236.354} C_VEL
LIN {X 0,Y 162.461,Z 643.09,A -85,B 0,C 180,E1 -23240.247,E2 -23240.247} C_VEL
LIN {X 0,Y 163.143,Z 635.348,A -85,B 0,C 180,E1 -23244.158,E2 -23244.158} C_VEL
LIN {X 0,Y 164.016,Z 627.333,A -85,B 0,C 180,E1 -23247.428,E2 -23247.428} C_VEL
LIN {X 0,Y 165.218,Z 617.558,A -85,B 0,C 180,E1 -23250.694,E2 -23250.694} C_VEL
LIN {X 0,Y 166.635,Z 606.81,A -85,B 0,C 180,E1 -23253.611,E2 -23253.611} C_VEL
LIN {X 0,Y 168.106,Z 594.952,A -85,B 0,C 180,E1 -23256.175,E2 -23256.175} C_VEL
LIN {X 0,Y 169.517,Z 583.239,A -85,B 0,C 180,E1 -23258.185,E2 -23258.185} C_VEL
LIN {X 0,Y 170.774,Z 570.774,A -85,B 0,C 180,E1 -23259.826,E2 -23259.826} C_VEL
LIN {X 0,Y 171.936,Z 556.02,A -85,B 0,C 180,E1 -23261.233,E2 -23261.233} C_VEL
LIN {X 0,Y 175.274,Z 495.88,A -85,B 0,C 180,E1 -23265.056,E2 -23265.056} C_VEL
LIN {X 0,Y 164.331,Z 463.015,A -85,B 0,C 180,E1 -23268.324,E2 -23268.324} C_VEL
LIN {X 0,Y 164.327,Z 463.011,A -85,B 0,C 180,E1 -23274.351,E2 -23274.351} C_VEL
LIN {X 0,Y 164.372,Z 463.009,A -85,B 0,C 180,E1 -23279.13,E2 -23279.13} C_VEL
LIN {X 0,Y 164.397,Z 463.006,A -85,B 0,C 180,E1 -23284.69,E2 -23284.69} C_VEL
LIN {X 0,Y 164.486,Z 462.994,A -85,B 0,C 180,E1 -23290.051,E2 -23290.051} C_VEL
LIN {X 0,Y 164.525,Z 462.99,A -85,B 0,C 180,E1 -23295.148,E2 -23295.148} C_VEL
LIN {X 0,Y 164.766,Z 462.956,A -85,B 0,C 180,E1 -23300.175,E2 -23300.175} C_VEL
LIN {X 0,Y 164.823,Z 462.954,A -85,B 0,C 180,E1 -23302.65,E2 -23302.65} C_VEL
LIN {X 0,Y 165.043,Z 462.923,A -85,B 0,C 180,E1 -23307.559,E2 -23307.559} C_VEL
LIN {X 0,Y 165.291,Z 462.89,A -85,B 0,C 180,E1 -23309.999,E2 -23309.999} C_VEL
LIN {X 0,Y 164.755,Z 462.961,A -85,B 0,C 180,E1 -23314.893,E2 -23314.893} C_VEL
LIN {X 0,Y 164.828,Z 462.947,A -85,B 0,C 180,E1 -23317.348,E2 -23317.348} C_VEL
LIN {X 0,Y 164.703,Z 462.968,A -85,B 0,C 180,E1 -23321.06,E2 -23321.06} C_VEL
LIN {X 0,Y 164.477,Z 462.992,A -85,B 0,C 180,E1 -23327.403,E2 -23327.403} C_VEL
LIN {X 0,Y 164.472,Z 462.996,A -85,B 0,C 180,E1 -23329.988,E2 -23329.988} C_VEL
LIN {X 0,Y 164.37,Z 463.005,A -85,B 0,C 180,E1 -23336.116,E2 -23336.116} C_VEL
LIN {X 0,Y 164.357,Z 463.01,A -85,B 0,C 180,E1 -23341.217,E2 -23341.217} C_VEL
LIN {X 0,Y 164.279,Z 463.022,A -85,B 0,C 180,E1 -23346.792,E2 -23346.792} C_VEL
LIN {X 0,Y 164.285,Z 463.02,A -85,B 0,C 180,E1 -23349.917,E2 -23349.917} C_VEL
LIN {X 0,Y 164.278,Z 463.017,A -85,B 0,C 180,E1 -23353.341,E2 -23353.341} C_VEL
LIN {X 0,Y 164.262,Z 463.024,A -85,B 0,C 180,E1 -23356.799,E2 -23356.799} C_VEL
LIN {X 0,Y 164.294,Z 463.017,A -85,B 0,C 180,E1 -23360.351,E2 -23360.351} C_VEL
LIN {X 0,Y 164.329,Z 463.014,A -85,B 0,C 180,E1 -23364.349,E2 -23364.349} C_VEL
LIN {X 0,Y 164.388,Z 463.003,A -85,B 0,C 180,E1 -23369.134,E2 -23369.134} C_VEL
LIN {X 0,Y 164.415,Z 463.006,A -85,B 0,C 180,E1 -23374.694,E2 -23374.694} C_VEL
LIN {X 0,Y 164.485,Z 462.991,A -85,B 0,C 180,E1 -23380.05,E2 -23380.05} C_VEL
LIN {X 0,Y 164.547,Z 462.986,A -85,B 0,C 180,E1 -23385.151,E2 -23385.151} C_VEL
LIN {X 0,Y 164.803,Z 462.954,A -85,B 0,C 180,E1 -23390.179,E2 -23390.179} C_VEL
LIN {X 0,Y 164.852,Z 462.951,A -85,B 0,C 180,E1 -23392.652,E2 -23392.652} C_VEL
LIN {X 0,Y 165.048,Z 462.922,A -85,B 0,C 180,E1 -23397.56,E2 -23397.56} C_VEL
LIN {X 0,Y 165.295,Z 462.894,A -85,B 0,C 180,E1 -23400,E2 -23400} C_VEL
LIN {X 0,Y 164.773,Z 462.955,A -85,B 0,C 180,E1 -23404.894,E2 -23404.894} C_VEL
LIN {X 0,Y 164.85,Z 462.949,A -85,B 0,C 180,E1 -23409.819,E2 -23409.819} C_VEL
LIN {X 0,Y 164.536,Z 462.986,A -85,B 0,C 180,E1 -23414.85,E2 -23414.85} C_VEL
LIN {X 0,Y 164.472,Z 462.996,A -85,B 0,C 180,E1 -23419.99,E2 -23419.99} C_VEL
LIN {X 0,Y 164.385,Z 463.007,A -85,B 0,C 180,E1 -23426.129,E2 -23426.129} C_VEL
LIN {X 0,Y 164.388,Z 463.003,A -85,B 0,C 180,E1 -23431.236,E2 -23431.236} C_VEL
LIN {X 0,Y 164.294,Z 463.02,A -85,B 0,C 180,E1 -23436.79,E2 -23436.79} C_VEL
LIN {X 0,Y 164.29,Z 463.014,A -85,B 0,C 180,E1 -23439.917,E2 -23439.917} C_VEL
LIN {X 0,Y 164.279,Z 463.021,A -85,B 0,C 180,E1 -23443.343,E2 -23443.343} C_VEL
LIN {X 0,Y 164.292,Z 463.018,A -85,B 0,C 180,E1 -23446.809,E2 -23446.809} C_VEL
LIN {X 0,Y 164.482,Z 463.193,A -85,B 0,C 180,E1 -23450.514,E2 -23450.514} C_VEL
LIN {X 0,Y 166.49,Z 473.019,A -85,B 0,C 180,E1 -23455.402,E2 -23455.402} C_VEL
LIN {X 0,Y 166.654,Z 473.881,A -85,B 0,C 180,E1 -23455.774,E2 -23455.774} C_VEL
LIN {X 0,Y 170.974,Z 491.005,A -85,B 0,C 180,E1 -23457.338,E2 -23457.338} C_VEL
LIN {X 0,Y 173.094,Z 525.175,A -85,B 0,C 180,E1 -23459.811,E2 -23459.811} C_VEL
LIN {X 0,Y 174.205,Z 540.086,A -85,B 0,C 180,E1 -23460.874,E2 -23460.874} C_VEL
LIN {X 0,Y 171.598,Z 585.066,A -85,B 0,C 180,E1 -23463.855,E2 -23463.855} C_VEL
LIN {X 0,Y 170.511,Z 598.152,A -85,B 0,C 180,E1 -23465.177,E2 -23465.177} C_VEL
LIN {X 0,Y 169.049,Z 610.362,A -85,B 0,C 180,E1 -23466.867,E2 -23466.867} C_VEL
LIN {X 0,Y 167.554,Z 622.8,A -85,B 0,C 180,E1 -23469.114,E2 -23469.114} C_VEL
LIN {X 0,Y 166.125,Z 634.446,A -85,B 0,C 180,E1 -23471.821,E2 -23471.821} C_VEL
LIN {X 0,Y 164.918,Z 643.884,A -85,B 0,C 180,E1 -23474.554,E2 -23474.554} C_VEL
LIN {X 0,Y 164.136,Z 652.603,A -85,B 0,C 180,E1 -23477.639,E2 -23477.639} C_VEL
LIN {X 0,Y 163.611,Z 660.469,A -85,B 0,C 180,E1 -23481.108,E2 -23481.108} C_VEL
LIN {X 0,Y 163.566,Z 666.617,A -85,B 0,C 180,E1 -23484.453,E2 -23484.453} C_VEL
LIN {X 0,Y 163.636,Z 671.207,A -85,B 0,C 180,E1 -23487.539,E2 -23487.539} C_VEL
LIN {X 0,Y 163.737,Z 674.15,A -85,B 0,C 180,E1 -23490.001,E2 -23490.001} C_VEL
LIN {X 0,Y 163.025,Z 677.475,A -85,B 0,C 180,E1 -23493.88,E2 -23493.88} C_VEL
LIN {X 0,Y 162.122,Z 678.693,A -85,B 0,C 180,E1 -23495.889,E2 -23495.889} C_VEL
LIN {X 0,Y 159.191,Z 679.759,A -85,B 0,C 180,E1 -23499.244,E2 -23499.244} C_VEL
LIN {X 0,Y 157.084,Z 680.183,A -85,B 0,C 180,E1 -23502.032,E2 -23502.032} C_VEL
LIN {X 0,Y 156.551,Z 680.474,A -85,B 0,C 180,E1 -23504.192,E2 -23504.192} C_VEL
LIN {X 0,Y 156.693,Z 680.55,A -85,B 0,C 180,E1 -23504.913,E2 -23504.913} C_VEL
LIN {X 0,Y 158.1,Z 680.737,A -85,B 0,C 180,E1 -23508.131,E2 -23508.131} C_VEL
LIN {X 0,Y 161.596,Z 679.849,A -85,B 0,C 180,E1 -23513.044,E2 -23513.044} C_VEL
LIN {X 0,Y 166.403,Z 677.611,A -85,B 0,C 180,E1 -23517.684,E2 -23517.684} C_VEL
LIN {X 0,Y 172.579,Z 673.997,A -85,B 0,C 180,E1 -23521.966,E2 -23521.966} C_VEL
LIN {X 0,Y 177.94,Z 670.29,A -85,B 0,C 180,E1 -23524.94,E2 -23524.94} C_VEL
LIN {X 0,Y 186.227,Z 663.921,A -85,B 0,C 180,E1 -23528.514,E2 -23528.514} C_VEL
LIN {X 0,Y 194.184,Z 656.829,A -85,B 0,C 180,E1 -23531.34,E2 -23531.34} C_VEL
LIN {X 0,Y 202.799,Z 648.095,A -85,B 0,C 180,E1 -23533.877,E2 -23533.877} C_VEL
LIN {X 0,Y 209.367,Z 640.599,A -85,B 0,C 180,E1 -23535.507,E2 -23535.507} C_VEL
LIN {X 0,Y 216.967,Z 630.743,A -85,B 0,C 180,E1 -23537.138,E2 -23537.138} C_VEL
LIN {X 0,Y 224.908,Z 618.872,A -85,B 0,C 180,E1 -23538.588,E2 -23538.588} C_VEL
LIN {X 0,Y 231.578,Z 606.982,A -85,B 0,C 180,E1 -23539.686,E2 -23539.686} C_VEL
LIN {X 0,Y 237.573,Z 593.902,A -85,B 0,C 180,E1 -23540.545,E2 -23540.545} C_VEL
LIN {X 0,Y 242.576,Z 580.403,A -85,B 0,C 180,E1 -23541.205,E2 -23541.205} C_VEL
LIN {X 0,Y 245.461,Z 570.398,A -85,B 0,C 180,E1 -23541.64,E2 -23541.64} C_VEL
LIN {X 0,Y 245.696,Z 568.454,A -85,B 0,C 180,E1 -23543.705,E2 -23543.705} C_VEL
LIN {X 0,Y 245.878,Z 568.155,A -85,B 0,C 180,E1 -23544.54,E2 -23544.54} C_VEL
LIN {X 0,Y 242.061,Z 580.969,A -85,B 0,C 180,E1 -23545.279,E2 -23545.279} C_VEL
LIN {X 0,Y 237.097,Z 593.611,A -85,B 0,C 180,E1 -23546.235,E2 -23546.235} C_VEL
LIN {X 0,Y 231.495,Z 605.168,A -85,B 0,C 180,E1 -23547.393,E2 -23547.393} C_VEL
LIN {X 0,Y 224.706,Z 616.587,A -85,B 0,C 180,E1 -23548.87,E2 -23548.87} C_VEL
LIN {X 0,Y 217.416,Z 626.782,A -85,B 0,C 180,E1 -23550.599,E2 -23550.599} C_VEL
LIN {X 0,Y 211.195,Z 634.302,A -85,B 0,C 180,E1 -23552.232,E2 -23552.232} C_VEL
LIN {X 0,Y 203.037,Z 642.713,A -85,B 0,C 180,E1 -23554.634,E2 -23554.634} C_VEL
LIN {X 0,Y 196.552,Z 648.508,A -85,B 0,C 180,E1 -23556.839,E2 -23556.839} C_VEL
LIN {X 0,Y 189.809,Z 653.612,A -85,B 0,C 180,E1 -23559.405,E2 -23559.405} C_VEL
LIN {X 0,Y 181.671,Z 658.652,A -85,B 0,C 180,E1 -23563.133,E2 -23563.133} C_VEL
LIN {X 0,Y 176.135,Z 661.289,A -85,B 0,C 180,E1 -23566.148,E2 -23566.148} C_VEL
LIN {X 0,Y 169.748,Z 663.367,A -85,B 0,C 180,E1 -23570.467,E2 -23570.467} C_VEL
LIN {X 0,Y 164.443,Z 663.828,A -85,B 0,C 180,E1 -23575.096,E2 -23575.096} C_VEL
LIN {X 0,Y 160.385,Z 662.754,A -85,B 0,C 180,E1 -23580,E2 -23580} C_VEL
LIN {X 0,Y 158.76,Z 661.619,A -85,B 0,C 180,E1 -23582.537,E2 -23582.537} C_VEL
LIN {X 0,Y 156.521,Z 658.099,A -85,B 0,C 180,E1 -23587.741,E2 -23587.741} C_VEL
LIN {X 0,Y 155.514,Z 654.3,A -85,B 0,C 180,E1 -23591.734,E2 -23591.734} C_VEL
LIN {X 0,Y 155.185,Z 649.367,A -85,B 0,C 180,E1 -23595.767,E2 -23595.767} C_VEL
LIN {X 0,Y 155.342,Z 643.134,A -85,B 0,C 180,E1 -23599.835,E2 -23599.835} C_VEL
LIN {X 0,Y 156.024,Z 635.33,A -85,B 0,C 180,E1 -23603.916,E2 -23603.916} C_VEL
LIN {X 0,Y 156.9,Z 627.243,A -85,B 0,C 180,E1 -23607.331,E2 -23607.331} C_VEL
LIN {X 0,Y 158.116,Z 617.34,A -85,B 0,C 180,E1 -23610.741,E2 -23610.741} C_VEL
LIN {X 0,Y 159.524,Z 606.632,A -85,B 0,C 180,E1 -23613.722,E2 -23613.722} C_VEL
LIN {X 0,Y 161.105,Z 594.259,A -85,B 0,C 180,E1 -23616.468,E2 -23616.468} C_VEL
LIN {X 0,Y 162.583,Z 581.954,A -85,B 0,C 180,E1 -23618.605,E2 -23618.605} C_VEL
LIN {X 0,Y 163.964,Z 568.21,A -85,B 0,C 180,E1 -23620.414,E2 -23620.414} C_VEL
LIN {X 0,Y 165.033,Z 554.202,A -85,B 0,C 180,E1 -23621.713,E2 -23621.713} C_VEL
LIN {X 0,Y 168.34,Z 497.286,A -85,B 0,C 180,E1 -23625.504,E2 -23625.504} C_VEL
LIN {X 0,Y 157.248,Z 463.897,A -85,B 0,C 180,E1 -23628.908,E2 -23628.908} C_VEL
LIN {X 0,Y 157.276,Z 463.889,A -85,B 0,C 180,E1 -23634.484,E2 -23634.484} C_VEL
LIN {X 0,Y 157.285,Z 463.893,A -85,B 0,C 180,E1 -23638.101,E2 -23638.101} C_VEL
LIN {X 0,Y 157.311,Z 463.884,A -85,B 0,C 180,E1 -23643.463,E2 -23643.463} C_VEL
LIN {X 0,Y 157.394,Z 463.877,A -85,B 0,C 180,E1 -23649.669,E2 -23649.669} C_VEL
LIN {X 0,Y 157.455,Z 463.871,A -85,B 0,C 180,E1 -23654.465,E2 -23654.465} C_VEL
LIN {X 0,Y 157.688,Z 463.838,A -85,B 0,C 180,E1 -23659.73,E2 -23659.73} C_VEL
LIN {X 0,Y 157.761,Z 463.831,A -85,B 0,C 180,E1 -23662.319,E2 -23662.319} C_VEL
LIN {X 0,Y 158.253,Z 463.767,A -85,B 0,C 180,E1 -23669.999,E2 -23669.999} C_VEL
LIN {X 0,Y 157.765,Z 463.826,A -85,B 0,C 180,E1 -23677.679,E2 -23677.679} C_VEL
LIN {X 0,Y 157.637,Z 463.848,A -85,B 0,C 180,E1 -23681.235,E2 -23681.235} C_VEL
LIN {X 0,Y 157.437,Z 463.869,A -85,B 0,C 180,E1 -23685.535,E2 -23685.535} C_VEL
LIN {X 0,Y 157.366,Z 463.883,A -85,B 0,C 180,E1 -23690.932,E2 -23690.932} C_VEL
LIN {X 0,Y 157.309,Z 463.887,A -85,B 0,C 180,E1 -23696.68,E2 -23696.68} C_VEL
LIN {X 0,Y 157.267,Z 463.892,A -85,B 0,C 180,E1 -23702.428,E2 -23702.428} C_VEL
LIN {X 0,Y 157.258,Z 463.895,A -85,B 0,C 180,E1 -23706.444,E2 -23706.444} C_VEL
LIN {X 0,Y 157.189,Z 463.901,A -85,B 0,C 180,E1 -23712.117,E2 -23712.117} C_VEL
LIN {X 0,Y 157.191,Z 463.904,A -85,B 0,C 180,E1 -23717.883,E2 -23717.883} C_VEL
LIN {X 0,Y 157.266,Z 463.892,A -85,B 0,C 180,E1 -23723.55,E2 -23723.55} C_VEL
LIN {X 0,Y 157.291,Z 463.891,A -85,B 0,C 180,E1 -23728.096,E2 -23728.096} C_VEL
LIN {X 0,Y 157.32,Z 463.887,A -85,B 0,C 180,E1 -23733.466,E2 -23733.466} C_VEL
LIN {X 0,Y 157.394,Z 463.874,A -85,B 0,C 180,E1 -23739.666,E2 -23739.666} C_VEL
LIN {X 0,Y 157.477,Z 463.87,A -85,B 0,C 180,E1 -23744.468,E2 -23744.468} C_VEL
LIN {X 0,Y 157.726,Z 463.835,A -85,B 0,C 180,E1 -23749.733,E2 -23749.733} C_VEL
LIN {X 0,Y 157.809,Z 463.828,A -85,B 0,C 180,E1 -23752.322,E2 -23752.322} C_VEL
LIN {X 0,Y 158.257,Z 463.771,A -85,B 0,C 180,E1 -23760,E2 -23760} C_VEL
LIN {X 0,Y 157.821,Z 463.824,A -85,B 0,C 180,E1 -23767.678,E2 -23767.678} C_VEL
LIN {X 0,Y 157.704,Z 463.838,A -85,B 0,C 180,E1 -23771.361,E2 -23771.361} C_VEL
LIN {X 0,Y 157.461,Z 463.868,A -85,B 0,C 180,E1 -23775.534,E2 -23775.534} C_VEL
LIN {X 0,Y 157.367,Z 463.879,A -85,B 0,C 180,E1 -23780.934,E2 -23780.934} C_VEL
LIN {X 0,Y 157.308,Z 463.891,A -85,B 0,C 180,E1 -23786.681,E2 -23786.681} C_VEL
LIN {X 0,Y 157.281,Z 463.889,A -85,B 0,C 180,E1 -23792.427,E2 -23792.427} C_VEL
LIN {X 0,Y 157.267,Z 463.896,A -85,B 0,C 180,E1 -23796.45,E2 -23796.45} C_VEL
LIN {X 0,Y 157.21,Z 463.899,A -85,B 0,C 180,E1 -23802.111,E2 -23802.111} C_VEL
LIN {X 0,Y 157.246,Z 463.893,A -85,B 0,C 180,E1 -23807.902,E2 -23807.902} C_VEL
LIN {X 0,Y 157.43,Z 463.975,A -85,B 0,C 180,E1 -23810.224,E2 -23810.224} C_VEL
LIN {X 0,Y 159.276,Z 473.12,A -85,B 0,C 180,E1 -23814.998,E2 -23814.998} C_VEL
LIN {X 0,Y 164.111,Z 492.179,A -85,B 0,C 180,E1 -23816.855,E2 -23816.855} C_VEL
LIN {X 0,Y 165.951,Z 523.162,A -85,B 0,C 180,E1 -23819.198,E2 -23819.198} C_VEL
LIN {X 0,Y 167.2,Z 540.376,A -85,B 0,C 180,E1 -23820.491,E2 -23820.491} C_VEL
LIN {X 0,Y 164.618,Z 583.998,A -85,B 0,C 180,E1 -23823.505,E2 -23823.505} C_VEL
LIN {X 0,Y 163.421,Z 598.06,A -85,B 0,C 180,E1 -23824.987,E2 -23824.987} C_VEL
LIN {X 0,Y 161.784,Z 611.537,A -85,B 0,C 180,E1 -23826.986,E2 -23826.986} C_VEL
LIN {X 0,Y 160.434,Z 622.698,A -85,B 0,C 180,E1 -23829.151,E2 -23829.151} C_VEL
LIN {X 0,Y 159.02,Z 634.158,A -85,B 0,C 180,E1 -23831.98,E2 -23831.98} C_VEL
LIN {X 0,Y 157.713,Z 644.424,A -85,B 0,C 180,E1 -23835.154,E2 -23835.154} C_VEL
LIN {X 0,Y 156.995,Z 652.863,A -85,B 0,C 180,E1 -23838.379,E2 -23838.379} C_VEL
LIN {X 0,Y 156.623,Z 660.061,A -85,B 0,C 180,E1 -23841.744,E2 -23841.744} C_VEL
LIN {X 0,Y 156.613,Z 665.568,A -85,B 0,C 180,E1 -23844.852,E2 -23844.852} C_VEL
LIN {X 0,Y 156.76,Z 671.01,A -85,B 0,C 180,E1 -23848.716,E2 -23848.716} C_VEL
LIN {X 0,Y 156.614,Z 673.775,A -85,B 0,C 180,E1 -23851.287,E2 -23851.287} C_VEL
LIN {X 0,Y 155.934,Z 676.839,A -85,B 0,C 180,E1 -23855.173,E2 -23855.173} C_VEL
LIN {X 0,Y 155.713,Z 679.47,A -85,B 0,C 180,E1 -23860.402,E2 -23860.402} C_VEL
LIN {X 0,Y 156.693,Z 680.55,A -85,B 0,C 180,E1 -23864.913,E2 -23864.913} C_VEL
LIN {X 0,Y 156.893,Z 680.704,A -85,B 0,C 180,E1 -23867.07,E2 -23867.07} C_VEL
LIN {X 0,Y 156.075,Z 680.28,A -85,B 0,C 180,E1 -23870.685,E2 -23870.685} C_VEL
LIN {X 0,Y 155.829,Z 679.573,A -85,B 0,C 180,E1 -23873.588,E2 -23873.588} C_VEL
LIN {X 0,Y 156.707,Z 678.935,A -85,B 0,C 180,E1 -23875.718,E2 -23875.718} C_VEL
LIN {X 0,Y 157.304,Z 678.694,A -85,B 0,C 180,E1 -23876.398,E2 -23876.398} C_VEL
LIN {X 0,Y 163.201,Z 676.119,A -85,B 0,C 180,E1 -23881.116,E2 -23881.116} C_VEL
LIN {X 0,Y 170.281,Z 672.14,A -85,B 0,C 180,E1 -23885.299,E2 -23885.299} C_VEL
LIN {X 0,Y 176.413,Z 668.225,A -85,B 0,C 180,E1 -23888.135,E2 -23888.135} C_VEL
LIN {X 0,Y 185.376,Z 661.49,A -85,B 0,C 180,E1 -23891.566,E2 -23891.566} C_VEL
LIN {X 0,Y 193.988,Z 654.139,A -85,B 0,C 180,E1 -23894.221,E2 -23894.221} C_VEL
LIN {X 0,Y 203.187,Z 644.942,A -85,B 0,C 180,E1 -23896.584,E2 -23896.584} C_VEL
LIN {X 0,Y 211.636,Z 635.392,A -85,B 0,C 180,E1 -23898.346,E2 -23898.346} C_VEL
LIN {X 0,Y 219.381,Z 625.191,A -85,B 0,C 180,E1 -23899.73,E2 -23899.73} C_VEL
LIN {X 0,Y 227.292,Z 612.88,A -85,B 0,C 180,E1 -23900.977,E2 -23900.977} C_VEL
LIN {X 0,Y 233.403,Z 601.644,A -85,B 0,C 180,E1 -23901.84,E2 -23901.84} C_VEL
LIN {X 0,Y 239.099,Z 588.776,A -85,B 0,C 180,E1 -23902.527,E2 -23902.527} C_VEL
LIN {X 0,Y 243.089,Z 577.483,A -85,B 0,C 180,E1 -23903.015,E2 -23903.015} C_VEL
LIN {X 0,Y 243.338,Z 576.579,A -85,B 0,C 180,E1 -23903.296,E2 -23903.296} C_VEL
LIN {X 0,Y 238.689,Z 589.413,A -85,B 0,C 180,E1 -23904.121,E2 -23904.121} C_VEL
LIN {X 0,Y 233.341,Z 600.919,A -85,B 0,C 180,E1 -23905.092,E2 -23905.092} C_VEL
LIN {X 0,Y 226.8,Z 612.294,A -85,B 0,C 180,E1 -23906.364,E2 -23906.364} C_VEL
LIN {X 0,Y 220.324,Z 621.888,A -85,B 0,C 180,E1 -23907.703,E2 -23907.703} C_VEL
LIN {X 0,Y 212.379,Z 631.708,A -85,B 0,C 180,E1 -23909.512,E2 -23909.512} C_VEL
LIN {X 0,Y 203.913,Z 640.585,A -85,B 0,C 180,E1 -23911.712,E2 -23911.712} C_VEL
LIN {X 0,Y 196.449,Z 647.195,A -85,B 0,C 180,E1 -23913.907,E2 -23913.907} C_VEL
LIN {X 0,Y 187.763,Z 653.62,A -85,B 0,C 180,E1 -23916.857,E2 -23916.857} C_VEL
LIN {X 0,Y 181.058,Z 657.751,A -85,B 0,C 180,E1 -23919.552,E2 -23919.552} C_VEL
LIN {X 0,Y 176.853,Z 659.935,A -85,B 0,C 180,E1 -23921.463,E2 -23921.463} C_VEL
LIN {X 0,Y 172.888,Z 661.671,A -85,B 0,C 180,E1 -23923.468,E2 -23923.468} C_VEL
LIN {X 0,Y 169.176,Z 662.996,A -85,B 0,C 180,E1 -23925.566,E2 -23925.566} C_VEL
LIN {X 0,Y 162.623,Z 664.456,A -85,B 0,C 180,E1 -23930.045,E2 -23930.045} C_VEL
LIN {X 0,Y 159.759,Z 664.612,A -85,B 0,C 180,E1 -23932.416,E2 -23932.416} C_VEL
LIN {X 0,Y 154.979,Z 663.717,A -85,B 0,C 180,E1 -23937.401,E2 -23937.401} C_VEL
LIN {X 0,Y 151.45,Z 661.307,A -85,B 0,C 180,E1 -23942.66,E2 -23942.66} C_VEL
LIN {X 0,Y 149.707,Z 658.391,A -85,B 0,C 180,E1 -23946.74,E2 -23946.74} C_VEL
LIN {X 0,Y 148.583,Z 654.486,A -85,B 0,C 180,E1 -23950.906,E2 -23950.906} C_VEL
LIN {X 0,Y 148.136,Z 649.491,A -85,B 0,C 180,E1 -23955.125,E2 -23955.125} C_VEL
LIN {X 0,Y 148.272,Z 643.147,A -85,B 0,C 180,E1 -23959.378,E2 -23959.378} C_VEL
LIN {X 0,Y 148.903,Z 635.167,A -85,B 0,C 180,E1 -23963.652,E2 -23963.652} C_VEL
LIN {X 0,Y 149.806,Z 626.991,A -85,B 0,C 180,E1 -23967.227,E2 -23967.227} C_VEL
LIN {X 0,Y 151.018,Z 617.047,A -85,B 0,C 180,E1 -23970.791,E2 -23970.791} C_VEL
LIN {X 0,Y 152.487,Z 606.064,A -85,B 0,C 180,E1 -23973.94,E2 -23973.94} C_VEL
LIN {X 0,Y 154.084,Z 593.618,A -85,B 0,C 180,E1 -23976.773,E2 -23976.773} C_VEL
LIN {X 0,Y 155.644,Z 580.933,A -85,B 0,C 180,E1 -23979.001,E2 -23979.001} C_VEL
LIN {X 0,Y 157.003,Z 567.182,A -85,B 0,C 180,E1 -23980.83,E2 -23980.83} C_VEL
LIN {X 0,Y 158.035,Z 552.795,A -85,B 0,C 180,E1 -23982.162,E2 -23982.162} C_VEL
LIN {X 0,Y 161.369,Z 498.687,A -85,B 0,C 180,E1 -23985.934,E2 -23985.934} C_VEL
LIN {X 0,Y 150.218,Z 464.772,A -85,B 0,C 180,E1 -23989.577,E2 -23989.577} C_VEL
LIN {X 0,Y 150.187,Z 464.773,A -85,B 0,C 180,E1 -23995.836,E2 -23995.836} C_VEL
LIN {X 0,Y 150.193,Z 464.775,A -85,B 0,C 180,E1 -23999.02,E2 -23999.02} C_VEL
LIN {X 0,Y 150.24,Z 464.765,A -85,B 0,C 180,E1 -24002.722,E2 -24002.722} C_VEL
LIN {X 0,Y 150.351,Z 464.754,A -85,B 0,C 180,E1 -24009.208,E2 -24009.208} C_VEL
LIN {X 0,Y 150.363,Z 464.752,A -85,B 0,C 180,E1 -24013.712,E2 -24013.712} C_VEL
LIN {X 0,Y 150.611,Z 464.719,A -85,B 0,C 180,E1 -24019.241,E2 -24019.241} C_VEL
LIN {X 0,Y 150.684,Z 464.711,A -85,B 0,C 180,E1 -24021.956,E2 -24021.956} C_VEL
LIN {X 0,Y 151.214,Z 464.643,A -85,B 0,C 180,E1 -24029.999,E2 -24029.999} C_VEL
LIN {X 0,Y 150.703,Z 464.706,A -85,B 0,C 180,E1 -24038.041,E2 -24038.041} C_VEL
LIN {X 0,Y 150.577,Z 464.727,A -85,B 0,C 180,E1 -24041.436,E2 -24041.436} C_VEL
LIN {X 0,Y 150.348,Z 464.752,A -85,B 0,C 180,E1 -24046.287,E2 -24046.287} C_VEL
LIN {X 0,Y 150.349,Z 464.757,A -85,B 0,C 180,E1 -24050.789,E2 -24050.789} C_VEL
LIN {X 0,Y 150.238,Z 464.768,A -85,B 0,C 180,E1 -24057.277,E2 -24057.277} C_VEL
LIN {X 0,Y 150.207,Z 464.77,A -85,B 0,C 180,E1 -24062.627,E2 -24062.627} C_VEL
LIN {X 0,Y 150.168,Z 464.778,A -85,B 0,C 180,E1 -24067.474,E2 -24067.474} C_VEL
LIN {X 0,Y 150.132,Z 464.779,A -85,B 0,C 180,E1 -24071.497,E2 -24071.497} C_VEL
LIN {X 0,Y 150.124,Z 464.783,A -85,B 0,C 180,E1 -24075.395,E2 -24075.395} C_VEL
LIN {X 0,Y 150.139,Z 464.78,A -85,B 0,C 180,E1 -24079.055,E2 -24079.055} C_VEL
LIN {X 0,Y 150.178,Z 464.774,A -85,B 0,C 180,E1 -24082.707,E2 -24082.707} C_VEL
LIN {X 0,Y 150.213,Z 464.772,A -85,B 0,C 180,E1 -24087.368,E2 -24087.368} C_VEL
LIN {X 0,Y 150.243,Z 464.77,A -85,B 0,C 180,E1 -24092.718,E2 -24092.718} C_VEL
LIN {X 0,Y 150.351,Z 464.751,A -85,B 0,C 180,E1 -24099.206,E2 -24099.206} C_VEL
LIN {X 0,Y 150.384,Z 464.751,A -85,B 0,C 180,E1 -24103.716,E2 -24103.716} C_VEL
LIN {X 0,Y 150.649,Z 464.717,A -85,B 0,C 180,E1 -24109.245,E2 -24109.245} C_VEL
LIN {X 0,Y 150.743,Z 464.707,A -85,B 0,C 180,E1 -24111.96,E2 -24111.96} C_VEL
LIN {X 0,Y 151.217,Z 464.648,A -85,B 0,C 180,E1 -24120,E2 -24120} C_VEL
LIN {X 0,Y 150.76,Z 464.704,A -85,B 0,C 180,E1 -24128.039,E2 -24128.039} C_VEL
LIN {X 0,Y 150.633,Z 464.719,A -85,B 0,C 180,E1 -24131.545,E2 -24131.545} C_VEL
LIN {X 0,Y 150.367,Z 464.752,A -85,B 0,C 180,E1 -24136.286,E2 -24136.286} C_VEL
LIN {X 0,Y 150.349,Z 464.754,A -85,B 0,C 180,E1 -24140.791,E2 -24140.791} C_VEL
LIN {X 0,Y 150.241,Z 464.77,A -85,B 0,C 180,E1 -24147.281,E2 -24147.281} C_VEL
LIN {X 0,Y 150.22,Z 464.769,A -85,B 0,C 180,E1 -24152.636,E2 -24152.636} C_VEL
LIN {X 0,Y 150.172,Z 464.776,A -85,B 0,C 180,E1 -24157.474,E2 -24157.474} C_VEL
LIN {X 0,Y 150.149,Z 464.778,A -85,B 0,C 180,E1 -24161.505,E2 -24161.505} C_VEL
LIN {X 0,Y 150.125,Z 464.783,A -85,B 0,C 180,E1 -24165.396,E2 -24165.396} C_VEL
LIN {X 0,Y 150.375,Z 464.94,A -85,B 0,C 180,E1 -24170.065,E2 -24170.065} C_VEL
LIN {X 0,Y 151.978,Z 472.68,A -85,B 0,C 180,E1 -24174.271,E2 -24174.271} C_VEL
LIN {X 0,Y 157.254,Z 494.002,A -85,B 0,C 180,E1 -24176.401,E2 -24176.401} C_VEL
LIN {X 0,Y 159.626,Z 532.589,A -85,B 0,C 180,E1 -24179.45,E2 -24179.45} C_VEL
LIN {X 0,Y 160.198,Z 540.473,A -85,B 0,C 180,E1 -24180.065,E2 -24180.065} C_VEL
LIN {X 0,Y 157.541,Z 584.011,A -85,B 0,C 180,E1 -24183.268,E2 -24183.268} C_VEL
LIN {X 0,Y 156.376,Z 597.523,A -85,B 0,C 180,E1 -24184.783,E2 -24184.783} C_VEL
LIN {X 0,Y 154.686,Z 611.204,A -85,B 0,C 180,E1 -24186.93,E2 -24186.93} C_VEL
LIN {X 0,Y 153.346,Z 622.315,A -85,B 0,C 180,E1 -24189.196,E2 -24189.196} C_VEL
LIN {X 0,Y 151.931,Z 633.725,A -85,B 0,C 180,E1 -24192.155,E2 -24192.155} C_VEL
LIN {X 0,Y 150.747,Z 643.004,A -85,B 0,C 180,E1 -24195.143,E2 -24195.143} C_VEL
LIN {X 0,Y 150.018,Z 651.607,A -85,B 0,C 180,E1 -24198.516,E2 -24198.516} C_VEL
LIN {X 0,Y 149.673,Z 659.914,A -85,B 0,C 180,E1 -24202.582,E2 -24202.582} C_VEL
LIN {X 0,Y 149.712,Z 665.455,A -85,B 0,C 180,E1 -24205.963,E2 -24205.963} C_VEL
LIN {X 0,Y 149.887,Z 670.682,A -85,B 0,C 180,E1 -24210.001,E2 -24210.001} C_VEL
LIN {X 0,Y 149.449,Z 673.279,A -85,B 0,C 180,E1 -24212.696,E2 -24212.696} C_VEL
LIN {X 0,Y 148.807,Z 676.577,A -85,B 0,C 180,E1 -24217.335,E2 -24217.335} C_VEL
LIN {X 0,Y 148.784,Z 678.269,A -85,B 0,C 180,E1 -24220.892,E2 -24220.892} C_VEL
LIN {X 0,Y 150.125,Z 679.733,A -85,B 0,C 180,E1 -24226.314,E2 -24226.314} C_VEL
LIN {X 0,Y 153.11,Z 679.864,A -85,B 0,C 180,E1 -24231.545,E2 -24231.545} C_VEL
LIN {X 0,Y 157.304,Z 678.694,A -85,B 0,C 180,E1 -24236.398,E2 -24236.398} C_VEL
LIN {X 0,Y 158.877,Z 677.947,A -85,B 0,C 180,E1 -24238.446,E2 -24238.446} C_VEL
LIN {X 0,Y 160.383,Z 676.257,A -85,B 0,C 180,E1 -24241.911,E2 -24241.911} C_VEL
LIN {X 0,Y 162.558,Z 673.986,A -85,B 0,C 180,E1 -24245.232,E2 -24245.232} C_VEL
LIN {X 0,Y 165.097,Z 672.331,A -85,B 0,C 180,E1 -24246.995,E2 -24246.995} C_VEL
LIN {X 0,Y 173.158,Z 667.646,A -85,B 0,C 180,E1 -24250.497,E2 -24250.497} C_VEL
LIN {X 0,Y 182.684,Z 661.071,A -85,B 0,C 180,E1 -24253.828,E2 -24253.828} C_VEL
LIN {X 0,Y 191.737,Z 653.774,A -85,B 0,C 180,E1 -24256.381,E2 -24256.381} C_VEL
LIN {X 0,Y 199.937,Z 646.268,A -85,B 0,C 180,E1 -24258.329,E2 -24258.329} C_VEL
LIN {X 0,Y 207.814,Z 638.03,A -85,B 0,C 180,E1 -24259.879,E2 -24259.879} C_VEL
LIN {X 0,Y 216.161,Z 628.011,A -85,B 0,C 180,E1 -24261.29,E2 -24261.29} C_VEL
LIN {X 0,Y 223.899,Z 617.166,A -85,B 0,C 180,E1 -24262.428,E2 -24262.428} C_VEL
LIN {X 0,Y 230.382,Z 606.404,A -85,B 0,C 180,E1 -24263.316,E2 -24263.316} C_VEL
LIN {X 0,Y 231.04,Z 605.172,A -85,B 0,C 180,E1 -24263.66,E2 -24263.66} C_VEL
LIN {X 0,Y 223.894,Z 616.537,A -85,B 0,C 180,E1 -24264.949,E2 -24264.949} C_VEL
LIN {X 0,Y 216.182,Z 626.682,A -85,B 0,C 180,E1 -24266.45,E2 -24266.45} C_VEL
LIN {X 0,Y 207.542,Z 636.23,A -85,B 0,C 180,E1 -24268.324,E2 -24268.324} C_VEL
LIN {X 0,Y 199.242,Z 643.95,A -85,B 0,C 180,E1 -24270.407,E2 -24270.407} C_VEL
LIN {X 0,Y 190.016,Z 651.137,A -85,B 0,C 180,E1 -24273.047,E2 -24273.047} C_VEL
LIN {X 0,Y 181.284,Z 656.681,A -85,B 0,C 180,E1 -24275.979,E2 -24275.979} C_VEL
LIN {X 0,Y 172.49,Z 661.103,A -85,B 0,C 180,E1 -24279.576,E2 -24279.576} C_VEL
LIN {X 0,Y 166,Z 663.498,A -85,B 0,C 180,E1 -24282.761,E2 -24282.761} C_VEL
LIN {X 0,Y 158.469,Z 665.134,A -85,B 0,C 180,E1 -24287.344,E2 -24287.344} C_VEL
LIN {X 0,Y 152.551,Z 665.213,A -85,B 0,C 180,E1 -24292.056,E2 -24292.056} C_VEL
LIN {X 0,Y 147.769,Z 663.781,A -85,B 0,C 180,E1 -24297.189,E2 -24297.189} C_VEL
LIN {X 0,Y 144.145,Z 660.743,A -85,B 0,C 180,E1 -24302.794,E2 -24302.794} C_VEL
LIN {X 0,Y 142.489,Z 657.482,A -85,B 0,C 180,E1 -24307.007,E2 -24307.007} C_VEL
LIN {X 0,Y 141.413,Z 653.024,A -85,B 0,C 180,E1 -24311.466,E2 -24311.466} C_VEL
LIN {X 0,Y 141.07,Z 646.441,A -85,B 0,C 180,E1 -24316.646,E2 -24316.646} C_VEL
LIN {X 0,Y 141.419,Z 639.265,A -85,B 0,C 180,E1 -24321.118,E2 -24321.118} C_VEL
LIN {X 0,Y 142.093,Z 631.856,A -85,B 0,C 180,E1 -24324.861,E2 -24324.861} C_VEL
LIN {X 0,Y 143.23,Z 622.253,A -85,B 0,C 180,E1 -24328.841,E2 -24328.841} C_VEL
LIN {X 0,Y 144.578,Z 611.806,A -85,B 0,C 180,E1 -24332.324,E2 -24332.324} C_VEL
LIN {X 0,Y 146.271,Z 599.412,A -85,B 0,C 180,E1 -24335.632,E2 -24335.632} C_VEL
LIN {X 0,Y 147.843,Z 587.223,A -85,B 0,C 180,E1 -24338.169,E2 -24338.169} C_VEL
LIN {X 0,Y 149.305,Z 573.772,A -85,B 0,C 180,E1 -24340.333,E2 -24340.333} C_VEL
LIN {X 0,Y 150.526,Z 560.158,A -85,B 0,C 180,E1 -24341.899,E2 -24341.899} C_VEL
LIN {X 0,Y 153.359,Z 515.889,A -85,B 0,C 180,E1 -24345.244,E2 -24345.244} C_VEL
LIN {X 0,Y 154.259,Z 499.501,A -85,B 0,C 180,E1 -24346.44,E2 -24346.44} C_VEL
LIN {X 0,Y 143.136,Z 465.656,A -85,B 0,C 180,E1 -24350.276,E2 -24350.276} C_VEL
LIN {X 0,Y 143.177,Z 465.649,A -85,B 0,C 180,E1 -24357.319,E2 -24357.319} C_VEL
LIN {X 0,Y 143.184,Z 465.645,A -85,B 0,C 180,E1 -24362.068,E2 -24362.068} C_VEL
LIN {X 0,Y 143.276,Z 465.636,A -85,B 0,C 180,E1 -24368.747,E2 -24368.747} C_VEL
LIN {X 0,Y 143.302,Z 465.632,A -85,B 0,C 180,E1 -24372.886,E2 -24372.886} C_VEL
LIN {X 0,Y 143.538,Z 465.601,A -85,B 0,C 180,E1 -24378.704,E2 -24378.704} C_VEL
LIN {X 0,Y 143.61,Z 465.592,A -85,B 0,C 180,E1 -24381.557,E2 -24381.557} C_VEL
LIN {X 0,Y 144.173,Z 465.52,A -85,B 0,C 180,E1 -24389.999,E2 -24389.999} C_VEL
LIN {X 0,Y 143.625,Z 465.589,A -85,B 0,C 180,E1 -24398.44,E2 -24398.44} C_VEL
LIN {X 0,Y 143.504,Z 465.608,A -85,B 0,C 180,E1 -24401.627,E2 -24401.627} C_VEL
LIN {X 0,Y 143.292,Z 465.631,A -85,B 0,C 180,E1 -24407.113,E2 -24407.113} C_VEL
LIN {X 0,Y 143.274,Z 465.637,A -85,B 0,C 180,E1 -24411.251,E2 -24411.251} C_VEL
LIN {X 0,Y 143.182,Z 465.647,A -85,B 0,C 180,E1 -24417.93,E2 -24417.93} C_VEL
LIN {X 0,Y 143.137,Z 465.649,A -85,B 0,C 180,E1 -24423.416,E2 -24423.416} C_VEL
LIN {X 0,Y 143.051,Z 465.664,A -85,B 0,C 180,E1 -24429.692,E2 -24429.692} C_VEL
LIN {X 0,Y 143.032,Z 465.663,A -85,B 0,C 180,E1 -24433.463,E2 -24433.463} C_VEL
LIN {X 0,Y 143.038,Z 465.667,A -85,B 0,C 180,E1 -24437.476,E2 -24437.476} C_VEL
LIN {X 0,Y 143.073,Z 465.656,A -85,B 0,C 180,E1 -24441.807,E2 -24441.807} C_VEL
LIN {X 0,Y 143.18,Z 465.648,A -85,B 0,C 180,E1 -24447.321,E2 -24447.321} C_VEL
LIN {X 0,Y 143.189,Z 465.645,A -85,B 0,C 180,E1 -24452.063,E2 -24452.063} C_VEL
LIN {X 0,Y 143.277,Z 465.632,A -85,B 0,C 180,E1 -24458.744,E2 -24458.744} C_VEL
LIN {X 0,Y 143.318,Z 465.633,A -85,B 0,C 180,E1 -24462.889,E2 -24462.889} C_VEL
LIN {X 0,Y 143.593,Z 465.594,A -85,B 0,C 180,E1 -24468.71,E2 -24468.71} C_VEL
LIN {X 0,Y 143.662,Z 465.589,A -85,B 0,C 180,E1 -24471.561,E2 -24471.561} C_VEL
LIN {X 0,Y 144.176,Z 465.525,A -85,B 0,C 180,E1 -24480,E2 -24480} C_VEL
LIN {X 0,Y 143.682,Z 465.587,A -85,B 0,C 180,E1 -24488.438,E2 -24488.438} C_VEL
LIN {X 0,Y 143.57,Z 465.598,A -85,B 0,C 180,E1 -24491.758,E2 -24491.758} C_VEL
LIN {X 0,Y 143.304,Z 465.634,A -85,B 0,C 180,E1 -24497.113,E2 -24497.113} C_VEL
LIN {X 0,Y 143.274,Z 465.633,A -85,B 0,C 180,E1 -24501.253,E2 -24501.253} C_VEL
LIN {X 0,Y 143.189,Z 465.648,A -85,B 0,C 180,E1 -24507.937,E2 -24507.937} C_VEL
LIN {X 0,Y 143.167,Z 465.649,A -85,B 0,C 180,E1 -24513.436,E2 -24513.436} C_VEL
LIN {X 0,Y 143.06,Z 465.658,A -85,B 0,C 180,E1 -24519.691,E2 -24519.691} C_VEL
LIN {X 0,Y 143.055,Z 465.664,A -85,B 0,C 180,E1 -24523.456,E2 -24523.456} C_VEL
LIN {X 0,Y 143.287,Z 465.729,A -85,B 0,C 180,E1 -24529.798,E2 -24529.798} C_VEL
LIN {X 0,Y 144.644,Z 472.055,A -85,B 0,C 180,E1 -24533.448,E2 -24533.448} C_VEL
LIN {X 0,Y 150.36,Z 494.78,A -85,B 0,C 180,E1 -24535.883,E2 -24535.883} C_VEL
LIN {X 0,Y 152.652,Z 533.226,A -85,B 0,C 180,E1 -24539.068,E2 -24539.068} C_VEL
LIN {X 0,Y 153.155,Z 540.744,A -85,B 0,C 180,E1 -24539.685,E2 -24539.685} C_VEL
LIN {X 0,Y 150.511,Z 583.608,A -85,B 0,C 180,E1 -24543.006,E2 -24543.006} C_VEL
LIN {X 0,Y 149.311,Z 597.129,A -85,B 0,C 180,E1 -24544.601,E2 -24544.601} C_VEL
LIN {X 0,Y 147.593,Z 610.865,A -85,B 0,C 180,E1 -24546.869,E2 -24546.869} C_VEL
LIN {X 0,Y 146.062,Z 623.277,A -85,B 0,C 180,E1 -24549.584,E2 -24549.584} C_VEL
LIN {X 0,Y 144.676,Z 634.414,A -85,B 0,C 180,E1 -24552.691,E2 -24552.691} C_VEL
LIN {X 0,Y 143.623,Z 643.446,A -85,B 0,C 180,E1 -24555.839,E2 -24555.839} C_VEL
LIN {X 0,Y 142.978,Z 651.902,A -85,B 0,C 180,E1 -24559.449,E2 -24559.449} C_VEL
LIN {X 0,Y 142.763,Z 659.833,A -85,B 0,C 180,E1 -24563.642,E2 -24563.642} C_VEL
LIN {X 0,Y 142.875,Z 665.245,A -85,B 0,C 180,E1 -24567.182,E2 -24567.182} C_VEL
LIN {X 0,Y 143.006,Z 668.803,A -85,B 0,C 180,E1 -24570.001,E2 -24570.001} C_VEL
LIN {X 0,Y 142.556,Z 671.597,A -85,B 0,C 180,E1 -24572.827,E2 -24572.827} C_VEL
LIN {X 0,Y 141.903,Z 675.203,A -85,B 0,C 180,E1 -24577.887,E2 -24577.887} C_VEL
LIN {X 0,Y 141.896,Z 676.956,A -85,B 0,C 180,E1 -24581.428,E2 -24581.428} C_VEL
LIN {X 0,Y 143.349,Z 678.743,A -85,B 0,C 180,E1 -24587.109,E2 -24587.109} C_VEL
LIN {X 0,Y 146.529,Z 679.206,A -85,B 0,C 180,E1 -24592.565,E2 -24592.565} C_VEL
LIN {X 0,Y 151.086,Z 678.317,A -85,B 0,C 180,E1 -24597.722,E2 -24597.722} C_VEL
LIN {X 0,Y 157.18,Z 676.133,A -85,B 0,C 180,E1 -24602.451,E2 -24602.451} C_VEL
LIN {X 0,Y 165.097,Z 672.331,A -85,B 0,C 180,E1 -24606.995,E2 -24606.995} C_VEL
LIN {X 0,Y 167.859,Z 670.58,A -85,B 0,C 180,E1 -24608.696,E2 -24608.696} C_VEL
LIN {X 0,Y 174.512,Z 664.894,A -85,B 0,C 180,E1 -24613.901,E2 -24613.901} C_VEL
LIN {X 0,Y 177.625,Z 662.532,A -85,B 0,C 180,E1 -24615.327,E2 -24615.327} C_VEL
LIN {X 0,Y 178.874,Z 661.665,A -85,B 0,C 180,E1 -24615.724,E2 -24615.724} C_VEL
LIN {X 0,Y 188.41,Z 654.706,A -85,B 0,C 180,E1 -24618.249,E2 -24618.249} C_VEL
LIN {X 0,Y 197.143,Z 647.23,A -85,B 0,C 180,E1 -24620.197,E2 -24620.197} C_VEL
LIN {X 0,Y 205.797,Z 638.887,A -85,B 0,C 180,E1 -24621.764,E2 -24621.764} C_VEL
LIN {X 0,Y 215.068,Z 628.411,A -85,B 0,C 180,E1 -24623.19,E2 -24623.19} C_VEL
LIN {X 0,Y 218.213,Z 624.389,A -85,B 0,C 180,E1 -24623.629,E2 -24623.629} C_VEL
LIN {X 0,Y 216.707,Z 626.132,A -85,B 0,C 180,E1 -24624.285,E2 -24624.285} C_VEL
LIN {X 0,Y 207.647,Z 635.959,A -85,B 0,C 180,E1 -24626.051,E2 -24626.051} C_VEL
LIN {X 0,Y 198.909,Z 643.83,A -85,B 0,C 180,E1 -24627.995,E2 -24627.995} C_VEL
LIN {X 0,Y 190.496,Z 650.283,A -85,B 0,C 180,E1 -24630.128,E2 -24630.128} C_VEL
LIN {X 0,Y 182.124,Z 655.616,A -85,B 0,C 180,E1 -24632.569,E2 -24632.569} C_VEL
LIN {X 0,Y 174.859,Z 659.481,A -85,B 0,C 180,E1 -24635.038,E2 -24635.038} C_VEL
LIN {X 0,Y 166.12,Z 663.088,A -85,B 0,C 180,E1 -24638.555,E2 -24638.555} C_VEL
LIN {X 0,Y 159.12,Z 665.095,A -85,B 0,C 180,E1 -24641.99,E2 -24641.99} C_VEL
LIN {X 0,Y 151.613,Z 666.072,A -85,B 0,C 180,E1 -24646.598,E2 -24646.598} C_VEL
LIN {X 0,Y 145.313,Z 665.584,A -85,B 0,C 180,E1 -24651.657,E2 -24651.657} C_VEL
LIN {X 0,Y 140.808,Z 663.814,A -85,B 0,C 180,E1 -24656.621,E2 -24656.621} C_VEL
LIN {X 0,Y 137.605,Z 661.016,A -85,B 0,C 180,E1 -24661.463,E2 -24661.463} C_VEL
LIN {X 0,Y 135.309,Z 656.436,A -85,B 0,C 180,E1 -24667.172,E2 -24667.172} C_VEL
LIN {X 0,Y 134.259,Z 651.319,A -85,B 0,C 180,E1 -24672.086,E2 -24672.086} C_VEL
LIN {X 0,Y 134.033,Z 645.209,A -85,B 0,C 180,E1 -24676.761,E2 -24676.761} C_VEL
LIN {X 0,Y 134.443,Z 637.636,A -85,B 0,C 180,E1 -24681.464,E2 -24681.464} C_VEL
LIN {X 0,Y 135.397,Z 628.129,A -85,B 0,C 180,E1 -24686.181,E2 -24686.181} C_VEL
LIN {X 0,Y 136.374,Z 619.809,A -85,B 0,C 180,E1 -24689.547,E2 -24689.547} C_VEL
LIN {X 0,Y 137.685,Z 609.914,A -85,B 0,C 180,E1 -24692.843,E2 -24692.843} C_VEL
LIN {X 0,Y 139.265,Z 598.622,A -85,B 0,C 180,E1 -24695.883,E2 -24695.883} C_VEL
LIN {X 0,Y 141.03,Z 584.998,A -85,B 0,C 180,E1 -24698.758,E2 -24698.758} C_VEL
LIN {X 0,Y 142.422,Z 571.887,A -85,B 0,C 180,E1 -24700.832,E2 -24700.832} C_VEL
LIN {X 0,Y 143.712,Z 557.748,A -85,B 0,C 180,E1 -24702.453,E2 -24702.453} C_VEL
LIN {X 0,Y 147.334,Z 501.05,A -85,B 0,C 180,E1 -24706.914,E2 -24706.914} C_VEL
LIN {X 0,Y 136.083,Z 466.54,A -85,B 0,C 180,E1 -24710.93,E2 -24710.93} C_VEL
LIN {X 0,Y 136.054,Z 466.533,A -85,B 0,C 180,E1 -24715.74,E2 -24715.74} C_VEL
LIN {X 0,Y 136.141,Z 466.521,A -85,B 0,C 180,E1 -24722.314,E2 -24722.314} C_VEL
LIN {X 0,Y 136.243,Z 466.512,A -85,B 0,C 180,E1 -24728.832,E2 -24728.832} C_VEL
LIN {X 0,Y 136.27,Z 466.51,A -85,B 0,C 180,E1 -24735.055,E2 -24735.055} C_VEL
LIN {X 0,Y 136.433,Z 466.489,A -85,B 0,C 180,E1 -24738.164,E2 -24738.164} C_VEL
LIN {X 0,Y 136.539,Z 466.473,A -85,B 0,C 180,E1 -24741.116,E2 -24741.116} C_VEL
LIN {X 0,Y 137.13,Z 466.397,A -85,B 0,C 180,E1 -24749.999,E2 -24749.999} C_VEL
LIN {X 0,Y 136.551,Z 466.472,A -85,B 0,C 180,E1 -24758.881,E2 -24758.881} C_VEL
LIN {X 0,Y 136.441,Z 466.489,A -85,B 0,C 180,E1 -24761.889,E2 -24761.889} C_VEL
LIN {X 0,Y 136.21,Z 466.514,A -85,B 0,C 180,E1 -24768.033,E2 -24768.033} C_VEL
LIN {X 0,Y 136.195,Z 466.519,A -85,B 0,C 180,E1 -24771.744,E2 -24771.744} C_VEL
LIN {X 0,Y 136.091,Z 466.533,A -85,B 0,C 180,E1 -24778.609,E2 -24778.609} C_VEL
LIN {X 0,Y 136.039,Z 466.534,A -85,B 0,C 180,E1 -24784.629,E2 -24784.629} C_VEL
LIN {X 0,Y 136.023,Z 466.54,A -85,B 0,C 180,E1 -24789.194,E2 -24789.194} C_VEL
LIN {X 0,Y 135.976,Z 466.542,A -85,B 0,C 180,E1 -24793.648,E2 -24793.648} C_VEL
LIN {X 0,Y 135.982,Z 466.546,A -85,B 0,C 180,E1 -24797.788,E2 -24797.788} C_VEL
LIN {X 0,Y 136.022,Z 466.534,A -85,B 0,C 180,E1 -24801.683,E2 -24801.683} C_VEL
LIN {X 0,Y 136.083,Z 466.533,A -85,B 0,C 180,E1 -24805.721,E2 -24805.721} C_VEL
LIN {X 0,Y 136.145,Z 466.523,A -85,B 0,C 180,E1 -24812.316,E2 -24812.316} C_VEL
LIN {X 0,Y 136.244,Z 466.508,A -85,B 0,C 180,E1 -24818.833,E2 -24818.833} C_VEL
LIN {X 0,Y 136.283,Z 466.507,A -85,B 0,C 180,E1 -24825.058,E2 -24825.058} C_VEL
LIN {X 0,Y 136.496,Z 466.475,A -85,B 0,C 180,E1 -24828.115,E2 -24828.115} C_VEL
LIN {X 0,Y 136.589,Z 466.471,A -85,B 0,C 180,E1 -24831.12,E2 -24831.12} C_VEL
LIN {X 0,Y 137.133,Z 466.402,A -85,B 0,C 180,E1 -24840,E2 -24840} C_VEL
LIN {X 0,Y 136.606,Z 466.469,A -85,B 0,C 180,E1 -24848.879,E2 -24848.879} C_VEL
LIN {X 0,Y 136.491,Z 466.48,A -85,B 0,C 180,E1 -24851.957,E2 -24851.957} C_VEL
LIN {X 0,Y 136.243,Z 466.513,A -85,B 0,C 180,E1 -24858.03,E2 -24858.03} C_VEL
LIN {X 0,Y 136.195,Z 466.514,A -85,B 0,C 180,E1 -24861.747,E2 -24861.747} C_VEL
LIN {X 0,Y 136.116,Z 466.529,A -85,B 0,C 180,E1 -24868.629,E2 -24868.629} C_VEL
LIN {X 0,Y 136.071,Z 466.535,A -85,B 0,C 180,E1 -24874.621,E2 -24874.621} C_VEL
LIN {X 0,Y 136.031,Z 466.534,A -85,B 0,C 180,E1 -24879.199,E2 -24879.199} C_VEL
LIN {X 0,Y 135.999,Z 466.543,A -85,B 0,C 180,E1 -24883.659,E2 -24883.659} C_VEL
LIN {X 0,Y 136.233,Z 466.612,A -85,B 0,C 180,E1 -24889.634,E2 -24889.634} C_VEL
LIN {X 0,Y 137.352,Z 471.817,A -85,B 0,C 180,E1 -24892.664,E2 -24892.664} C_VEL
LIN {X 0,Y 143.497,Z 496.233,A -85,B 0,C 180,E1 -24895.373,E2 -24895.373} C_VEL
LIN {X 0,Y 145.635,Z 533.305,A -85,B 0,C 180,E1 -24898.61,E2 -24898.61} C_VEL
LIN {X 0,Y 146.138,Z 541.076,A -85,B 0,C 180,E1 -24899.282,E2 -24899.282} C_VEL
LIN {X 0,Y 143.488,Z 582.741,A -85,B 0,C 180,E1 -24902.67,E2 -24902.67} C_VEL
LIN {X 0,Y 142.267,Z 596.606,A -85,B 0,C 180,E1 -24904.391,E2 -24904.391} C_VEL
LIN {X 0,Y 140.525,Z 610.376,A -85,B 0,C 180,E1 -24906.807,E2 -24906.807} C_VEL
LIN {X 0,Y 139,Z 622.672,A -85,B 0,C 180,E1 -24909.66,E2 -24909.66} C_VEL
LIN {X 0,Y 137.626,Z 633.708,A -85,B 0,C 180,E1 -24912.926,E2 -24912.926} C_VEL
LIN {X 0,Y 136.526,Z 643.643,A -85,B 0,C 180,E1 -24916.607,E2 -24916.607} C_VEL
LIN {X 0,Y 135.991,Z 651.364,A -85,B 0,C 180,E1 -24920.11,E2 -24920.11} C_VEL
LIN {X 0,Y 135.876,Z 658.546,A -85,B 0,C 180,E1 -24924.063,E2 -24924.063} C_VEL
LIN {X 0,Y 136.064,Z 665.009,A -85,B 0,C 180,E1 -24928.521,E2 -24928.521} C_VEL
LIN {X 0,Y 136.021,Z 668.366,A -85,B 0,C 180,E1 -24931.481,E2 -24931.481} C_VEL
LIN {X 0,Y 135.226,Z 672.088,A -85,B 0,C 180,E1 -24935.967,E2 -24935.967} C_VEL
LIN {X 0,Y 134.975,Z 674.044,A -85,B 0,C 180,E1 -24938.988,E2 -24938.988} C_VEL
LIN {X 0,Y 135.621,Z 676.779,A -85,B 0,C 180,E1 -24945.018,E2 -24945.018} C_VEL
LIN {X 0,Y 138.051,Z 678.18,A -85,B 0,C 180,E1 -24950.878,E2 -24950.878} C_VEL
LIN {X 0,Y 142.222,Z 678.303,A -85,B 0,C 180,E1 -24956.408,E2 -24956.408} C_VEL
LIN {X 0,Y 147.861,Z 677.147,A -85,B 0,C 180,E1 -24961.524,E2 -24961.524} C_VEL
LIN {X 0,Y 154.944,Z 674.73,A -85,B 0,C 180,E1 -24966.134,E2 -24966.134} C_VEL
LIN {X 0,Y 163.246,Z 670.936,A -85,B 0,C 180,E1 -24970.225,E2 -24970.225} C_VEL
LIN {X 0,Y 172.704,Z 665.682,A -85,B 0,C 180,E1 -24973.774,E2 -24973.774} C_VEL
LIN {X 0,Y 178.874,Z 661.665,A -85,B 0,C 180,E1 -24975.724,E2 -24975.724} C_VEL
LIN {X 0,Y 182.433,Z 659.086,A -85,B 0,C 180,E1 -24976.985,E2 -24976.985} C_VEL
LIN {X 0,Y 187.329,Z 654.952,A -85,B 0,C 180,E1 -24979.346,E2 -24979.346} C_VEL
LIN {X 0,Y 192.416,Z 650.344,A -85,B 0,C 180,E1 -24981.479,E2 -24981.479} C_VEL
LIN {X 0,Y 196.141,Z 647.038,A -85,B 0,C 180,E1 -24982.386,E2 -24982.386} C_VEL
LIN {X 0,Y 204.696,Z 639.114,A -85,B 0,C 180,E1 -24983.79,E2 -24983.79} C_VEL
LIN {X 0,Y 205.083,Z 638.633,A -85,B 0,C 180,E1 -24984.368,E2 -24984.368} C_VEL
LIN {X 0,Y 196.92,Z 645.51,A -85,B 0,C 180,E1 -24986.05,E2 -24986.05} C_VEL
LIN {X 0,Y 187.285,Z 652.296,A -85,B 0,C 180,E1 -24988.307,E2 -24988.307} C_VEL
LIN {X 0,Y 178.887,Z 657.214,A -85,B 0,C 180,E1 -24990.587,E2 -24990.587} C_VEL
LIN {X 0,Y 170.933,Z 660.991,A -85,B 0,C 180,E1 -24993.11,E2 -24993.11} C_VEL
LIN {X 0,Y 161.072,Z 664.526,A -85,B 0,C 180,E1 -24996.877,E2 -24996.877} C_VEL
LIN {X 0,Y 152.236,Z 666.447,A -85,B 0,C 180,E1 -25001.146,E2 -25001.146} C_VEL
LIN {X 0,Y 144.527,Z 666.821,A -85,B 0,C 180,E1 -25005.928,E2 -25005.928} C_VEL
LIN {X 0,Y 138.076,Z 665.723,A -85,B 0,C 180,E1 -25011.216,E2 -25011.216} C_VEL
LIN {X 0,Y 133.131,Z 663.113,A -85,B 0,C 180,E1 -25016.974,E2 -25016.974} C_VEL
LIN {X 0,Y 129.586,Z 658.933,A -85,B 0,C 180,E1 -25023.109,E2 -25023.109} C_VEL
LIN {X 0,Y 127.891,Z 654.122,A -85,B 0,C 180,E1 -25028.438,E2 -25028.438} C_VEL
LIN {X 0,Y 127.074,Z 648.295,A -85,B 0,C 180,E1 -25033.594,E2 -25033.594} C_VEL
LIN {X 0,Y 127.13,Z 641.398,A -85,B 0,C 180,E1 -25038.534,E2 -25038.534} C_VEL
LIN {X 0,Y 127.783,Z 632.725,A -85,B 0,C 180,E1 -25043.5,E2 -25043.5} C_VEL
LIN {X 0,Y 128.74,Z 623.834,A -85,B 0,C 180,E1 -25047.647,E2 -25047.647} C_VEL
LIN {X 0,Y 130.161,Z 612.912,A -85,B 0,C 180,E1 -25051.765,E2 -25051.765} C_VEL
LIN {X 0,Y 131.845,Z 600.693,A -85,B 0,C 180,E1 -25055.429,E2 -25055.429} C_VEL
LIN {X 0,Y 133.512,Z 588.145,A -85,B 0,C 180,E1 -25058.329,E2 -25058.329} C_VEL
LIN {X 0,Y 134.995,Z 575.413,A -85,B 0,C 180,E1 -25060.599,E2 -25060.599} C_VEL
LIN {X 0,Y 136.343,Z 561.571,A -85,B 0,C 180,E1 -25062.395,E2 -25062.395} C_VEL
LIN {X 0,Y 137.993,Z 536.245,A -85,B 0,C 180,E1 -25064.615,E2 -25064.615} C_VEL
LIN {X 0,Y 140.285,Z 502.105,A -85,B 0,C 180,E1 -25067.395,E2 -25067.395} C_VEL
LIN {X 0,Y 129.044,Z 467.409,A -85,B 0,C 180,E1 -25071.719,E2 -25071.719} C_VEL
LIN {X 0,Y 128.973,Z 467.419,A -85,B 0,C 180,E1 -25076.979,E2 -25076.979} C_VEL
LIN {X 0,Y 129.018,Z 467.411,A -85,B 0,C 180,E1 -25080.641,E2 -25080.641} C_VEL
LIN {X 0,Y 129.109,Z 467.402,A -85,B 0,C 180,E1 -25087.6,E2 -25087.6} C_VEL
LIN {X 0,Y 129.153,Z 467.39,A -85,B 0,C 180,E1 -25090.943,E2 -25090.943} C_VEL
LIN {X 0,Y 129.39,Z 467.366,A -85,B 0,C 180,E1 -25097.875,E2 -25097.875} C_VEL
LIN {X 0,Y 129.465,Z 467.352,A -85,B 0,C 180,E1 -25100.626,E2 -25100.626} C_VEL
LIN {X 0,Y 130.085,Z 467.275,A -85,B 0,C 180,E1 -25109.999,E2 -25109.999} C_VEL
LIN {X 0,Y 129.474,Z 467.354,A -85,B 0,C 180,E1 -25119.371,E2 -25119.371} C_VEL
LIN {X 0,Y 129.344,Z 467.374,A -85,B 0,C 180,E1 -25122.552,E2 -25122.552} C_VEL
LIN {X 0,Y 129.131,Z 467.399,A -85,B 0,C 180,E1 -25129.058,E2 -25129.058} C_VEL
LIN {X 0,Y 129.107,Z 467.402,A -85,B 0,C 180,E1 -25132.397,E2 -25132.397} C_VEL
LIN {X 0,Y 129.016,Z 467.414,A -85,B 0,C 180,E1 -25139.357,E2 -25139.357} C_VEL
LIN {X 0,Y 128.955,Z 467.418,A -85,B 0,C 180,E1 -25145.165,E2 -25145.165} C_VEL
LIN {X 0,Y 128.921,Z 467.422,A -85,B 0,C 180,E1 -25150.855,E2 -25150.855} C_VEL
LIN {X 0,Y 128.91,Z 467.426,A -85,B 0,C 180,E1 -25155.131,E2 -25155.131} C_VEL
LIN {X 0,Y 128.934,Z 467.421,A -85,B 0,C 180,E1 -25159.738,E2 -25159.738} C_VEL
LIN {X 0,Y 128.979,Z 467.419,A -85,B 0,C 180,E1 -25164.818,E2 -25164.818} C_VEL
LIN {X 0,Y 129.015,Z 467.408,A -85,B 0,C 180,E1 -25170.642,E2 -25170.642} C_VEL
LIN {X 0,Y 129.029,Z 467.412,A -85,B 0,C 180,E1 -25174.167,E2 -25174.167} C_VEL
LIN {X 0,Y 129.106,Z 467.398,A -85,B 0,C 180,E1 -25177.727,E2 -25177.727} C_VEL
LIN {X 0,Y 129.161,Z 467.394,A -85,B 0,C 180,E1 -25180.945,E2 -25180.945} C_VEL
LIN {X 0,Y 129.415,Z 467.356,A -85,B 0,C 180,E1 -25187.82,E2 -25187.82} C_VEL
LIN {X 0,Y 129.515,Z 467.351,A -85,B 0,C 180,E1 -25190.631,E2 -25190.631} C_VEL
LIN {X 0,Y 130.088,Z 467.28,A -85,B 0,C 180,E1 -25200,E2 -25200} C_VEL
LIN {X 0,Y 129.529,Z 467.35,A -85,B 0,C 180,E1 -25209.368,E2 -25209.368} C_VEL
LIN {X 0,Y 129.392,Z 467.363,A -85,B 0,C 180,E1 -25212.549,E2 -25212.549} C_VEL
LIN {X 0,Y 129.153,Z 467.396,A -85,B 0,C 180,E1 -25219.057,E2 -25219.057} C_VEL
LIN {X 0,Y 129.107,Z 467.397,A -85,B 0,C 180,E1 -25222.399,E2 -25222.399} C_VEL
LIN {X 0,Y 129.035,Z 467.408,A -85,B 0,C 180,E1 -25229.374,E2 -25229.374} C_VEL
LIN {X 0,Y 128.981,Z 467.418,A -85,B 0,C 180,E1 -25235.184,E2 -25235.184} C_VEL
LIN {X 0,Y 128.933,Z 467.419,A -85,B 0,C 180,E1 -25240.852,E2 -25240.852} C_VEL
LIN {X 0,Y 128.945,Z 467.422,A -85,B 0,C 180,E1 -25245.118,E2 -25245.118} C_VEL
LIN {X 0,Y 129.144,Z 467.43,A -85,B 0,C 180,E1 -25249.42,E2 -25249.42} C_VEL
LIN {X 0,Y 129.934,Z 471.064,A -85,B 0,C 180,E1 -25251.734,E2 -25251.734} C_VEL
LIN {X 0,Y 136.615,Z 497.576,A -85,B 0,C 180,E1 -25254.853,E2 -25254.853} C_VEL
LIN {X 0,Y 138.602,Z 533.459,A -85,B 0,C 180,E1 -25258.153,E2 -25258.153} C_VEL
LIN {X 0,Y 139.072,Z 541.854,A -85,B 0,C 180,E1 -25258.91,E2 -25258.91} C_VEL
LIN {X 0,Y 136.474,Z 581.929,A -85,B 0,C 180,E1 -25262.39,E2 -25262.39} C_VEL
LIN {X 0,Y 135.238,Z 595.792,A -85,B 0,C 180,E1 -25264.201,E2 -25264.201} C_VEL
LIN {X 0,Y 133.488,Z 609.616,A -85,B 0,C 180,E1 -25266.743,E2 -25266.743} C_VEL
LIN {X 0,Y 131.942,Z 621.936,A -85,B 0,C 180,E1 -25269.744,E2 -25269.744} C_VEL
LIN {X 0,Y 130.589,Z 632.994,A -85,B 0,C 180,E1 -25273.187,E2 -25273.187} C_VEL
LIN {X 0,Y 129.602,Z 642.043,A -85,B 0,C 180,E1 -25276.677,E2 -25276.677} C_VEL
LIN {X 0,Y 129.043,Z 650.35,A -85,B 0,C 180,E1 -25280.598,E2 -25280.598} C_VEL
LIN {X 0,Y 129.03,Z 658.352,A -85,B 0,C 180,E1 -25285.315,E2 -25285.315} C_VEL
LIN {X 0,Y 129.296,Z 664.612,A -85,B 0,C 180,E1 -25290.001,E2 -25290.001} C_VEL
LIN {X 0,Y 128.918,Z 667.782,A -85,B 0,C 180,E1 -25293.126,E2 -25293.126} C_VEL
LIN {X 0,Y 128.368,Z 670.315,A -85,B 0,C 180,E1 -25296.288,E2 -25296.288} C_VEL
LIN {X 0,Y 128.249,Z 674.051,A -85,B 0,C 180,E1 -25302.663,E2 -25302.663} C_VEL
LIN {X 0,Y 129.937,Z 676.443,A -85,B 0,C 180,E1 -25308.938,E2 -25308.938} C_VEL
LIN {X 0,Y 133.535,Z 677.54,A -85,B 0,C 180,E1 -25314.902,E2 -25314.902} C_VEL
LIN {X 0,Y 139.018,Z 677.334,A -85,B 0,C 180,E1 -25320.747,E2 -25320.747} C_VEL
LIN {X 0,Y 145.386,Z 675.966,A -85,B 0,C 180,E1 -25325.458,E2 -25325.458} C_VEL
LIN {X 0,Y 153.434,Z 673.274,A -85,B 0,C 180,E1 -25329.888,E2 -25329.888} C_VEL
LIN {X 0,Y 162.704,Z 669.243,A -85,B 0,C 180,E1 -25333.72,E2 -25333.72} C_VEL
LIN {X 0,Y 172.865,Z 663.794,A -85,B 0,C 180,E1 -25337.039,E2 -25337.039} C_VEL
LIN {X 0,Y 181.036,Z 658.585,A -85,B 0,C 180,E1 -25339.203,E2 -25339.203} C_VEL
LIN {X 0,Y 191.183,Z 651.147,A -85,B 0,C 180,E1 -25341.453,E2 -25341.453} C_VEL
LIN {X 0,Y 196.141,Z 647.038,A -85,B 0,C 180,E1 -25342.386,E2 -25342.386} C_VEL
LIN {X 0,Y 196.526,Z 646.613,A -85,B 0,C 180,E1 -25342.681,E2 -25342.681} C_VEL
LIN {X 0,Y 195.952,Z 646.838,A -85,B 0,C 180,E1 -25343.327,E2 -25343.327} C_VEL
LIN {X 0,Y 193.994,Z 648.105,A -85,B 0,C 180,E1 -25344.157,E2 -25344.157} C_VEL
LIN {X 0,Y 188.096,Z 652.025,A -85,B 0,C 180,E1 -25345.575,E2 -25345.575} C_VEL
LIN {X 0,Y 182.82,Z 655.151,A -85,B 0,C 180,E1 -25346.774,E2 -25346.774} C_VEL
LIN {X 0,Y 175.522,Z 658.939,A -85,B 0,C 180,E1 -25348.632,E2 -25348.632} C_VEL
LIN {X 0,Y 167.241,Z 662.501,A -85,B 0,C 180,E1 -25351.101,E2 -25351.101} C_VEL
LIN {X 0,Y 159.41,Z 665.06,A -85,B 0,C 180,E1 -25353.84,E2 -25353.84} C_VEL
LIN {X 0,Y 149.779,Z 667.116,A -85,B 0,C 180,E1 -25357.952,E2 -25357.952} C_VEL
LIN {X 0,Y 141.25,Z 667.628,A -85,B 0,C 180,E1 -25362.63,E2 -25362.63} C_VEL
LIN {X 0,Y 133.998,Z 666.65,A -85,B 0,C 180,E1 -25367.889,E2 -25367.889} C_VEL
LIN {X 0,Y 128.164,Z 664.232,A -85,B 0,C 180,E1 -25373.703,E2 -25373.703} C_VEL
LIN {X 0,Y 123.868,Z 660.224,A -85,B 0,C 180,E1 -25380,E2 -25380} C_VEL
LIN {X 0,Y 121.22,Z 654.622,A -85,B 0,C 180,E1 -25386.658,E2 -25386.658} C_VEL
LIN {X 0,Y 120.135,Z 648.037,A -85,B 0,C 180,E1 -25392.672,E2 -25392.672} C_VEL
LIN {X 0,Y 120.179,Z 639.687,A -85,B 0,C 180,E1 -25398.762,E2 -25398.762} C_VEL
LIN {X 0,Y 120.874,Z 630.608,A -85,B 0,C 180,E1 -25404.017,E2 -25404.017} C_VEL
LIN {X 0,Y 122.043,Z 620.214,A -85,B 0,C 180,E1 -25408.78,E2 -25408.78} C_VEL
LIN {X 0,Y 123.453,Z 609.436,A -85,B 0,C 180,E1 -25412.739,E2 -25412.739} C_VEL
LIN {X 0,Y 125.112,Z 597.843,A -85,B 0,C 180,E1 -25416.144,E2 -25416.144} C_VEL
LIN {X 0,Y 126.834,Z 584.884,A -85,B 0,C 180,E1 -25419.125,E2 -25419.125} C_VEL
LIN {X 0,Y 128.423,Z 570.672,A -85,B 0,C 180,E1 -25421.571,E2 -25421.571} C_VEL
LIN {X 0,Y 129.721,Z 556.34,A -85,B 0,C 180,E1 -25423.29,E2 -25423.29} C_VEL
LIN {X 0,Y 133.256,Z 503.259,A -85,B 0,C 180,E1 -25427.922,E2 -25427.922} C_VEL
LIN {X 0,Y 121.95,Z 468.29,A -85,B 0,C 180,E1 -25432.518,E2 -25432.518} C_VEL
LIN {X 0,Y 121.899,Z 468.301,A -85,B 0,C 180,E1 -25438.741,E2 -25438.741} C_VEL
LIN {X 0,Y 121.94,Z 468.289,A -85,B 0,C 180,E1 -25442.542,E2 -25442.542} C_VEL
LIN {X 0,Y 122.029,Z 468.284,A -85,B 0,C 180,E1 -25447.145,E2 -25447.145} C_VEL
LIN {X 0,Y 122.109,Z 468.271,A -85,B 0,C 180,E1 -25453.274,E2 -25453.274} C_VEL
LIN {X 0,Y 122.313,Z 468.248,A -85,B 0,C 180,E1 -25457.636,E2 -25457.636} C_VEL
LIN {X 0,Y 122.415,Z 468.235,A -85,B 0,C 180,E1 -25463.405,E2 -25463.405} C_VEL
LIN {X 0,Y 123.038,Z 468.152,A -85,B 0,C 180,E1 -25469.999,E2 -25469.999} C_VEL
LIN {X 0,Y 122.421,Z 468.23,A -85,B 0,C 180,E1 -25476.592,E2 -25476.592} C_VEL
LIN {X 0,Y 122.322,Z 468.249,A -85,B 0,C 180,E1 -25482.385,E2 -25482.385} C_VEL
LIN {X 0,Y 122.094,Z 468.27,A -85,B 0,C 180,E1 -25486.726,E2 -25486.726} C_VEL
LIN {X 0,Y 122.026,Z 468.282,A -85,B 0,C 180,E1 -25492.853,E2 -25492.853} C_VEL
LIN {X 0,Y 121.938,Z 468.293,A -85,B 0,C 180,E1 -25497.456,E2 -25497.456} C_VEL
LIN {X 0,Y 121.897,Z 468.299,A -85,B 0,C 180,E1 -25501.257,E2 -25501.257} C_VEL
LIN {X 0,Y 121.879,Z 468.3,A -85,B 0,C 180,E1 -25506.168,E2 -25506.168} C_VEL
LIN {X 0,Y 121.861,Z 468.3,A -85,B 0,C 180,E1 -25511.433,E2 -25511.433} C_VEL
LIN {X 0,Y 121.862,Z 468.304,A -85,B 0,C 180,E1 -25518.565,E2 -25518.565} C_VEL
LIN {X 0,Y 121.931,Z 468.297,A -85,B 0,C 180,E1 -25524.803,E2 -25524.803} C_VEL
LIN {X 0,Y 121.927,Z 468.29,A -85,B 0,C 180,E1 -25529.837,E2 -25529.837} C_VEL
LIN {X 0,Y 121.982,Z 468.29,A -85,B 0,C 180,E1 -25536.215,E2 -25536.215} C_VEL
LIN {X 0,Y 122.049,Z 468.276,A -85,B 0,C 180,E1 -25539.788,E2 -25539.788} C_VEL
LIN {X 0,Y 122.263,Z 468.249,A -85,B 0,C 180,E1 -25546.707,E2 -25546.707} C_VEL
LIN {X 0,Y 122.445,Z 468.23,A -85,B 0,C 180,E1 -25550.085,E2 -25550.085} C_VEL
LIN {X 0,Y 122.604,Z 468.206,A -85,B 0,C 180,E1 -25556.714,E2 -25556.714} C_VEL
LIN {X 0,Y 123.042,Z 468.157,A -85,B 0,C 180,E1 -25560,E2 -25560} C_VEL
LIN {X 0,Y 122.453,Z 468.227,A -85,B 0,C 180,E1 -25566.592,E2 -25566.592} C_VEL
LIN {X 0,Y 122.455,Z 468.231,A -85,B 0,C 180,E1 -25569.915,E2 -25569.915} C_VEL
LIN {X 0,Y 122.261,Z 468.248,A -85,B 0,C 180,E1 -25573.293,E2 -25573.293} C_VEL
LIN {X 0,Y 122.045,Z 468.282,A -85,B 0,C 180,E1 -25580.213,E2 -25580.213} C_VEL
LIN {X 0,Y 121.981,Z 468.286,A -85,B 0,C 180,E1 -25583.785,E2 -25583.785} C_VEL
LIN {X 0,Y 121.941,Z 468.291,A -85,B 0,C 180,E1 -25590.174,E2 -25590.174} C_VEL
LIN {X 0,Y 121.898,Z 468.301,A -85,B 0,C 180,E1 -25596.182,E2 -25596.182} C_VEL
LIN {X 0,Y 121.874,Z 468.301,A -85,B 0,C 180,E1 -25601.441,E2 -25601.441} C_VEL
LIN {X 0,Y 122.095,Z 468.334,A -85,B 0,C 180,E1 -25609.323,E2 -25609.323} C_VEL
LIN {X 0,Y 122.643,Z 470.622,A -85,B 0,C 180,E1 -25610.796,E2 -25610.796} C_VEL
LIN {X 0,Y 129.705,Z 498.504,A -85,B 0,C 180,E1 -25614.288,E2 -25614.288} C_VEL
LIN {X 0,Y 131.63,Z 534.362,A -85,B 0,C 180,E1 -25617.773,E2 -25617.773} C_VEL
LIN {X 0,Y 132.02,Z 542.176,A -85,B 0,C 180,E1 -25618.521,E2 -25618.521} C_VEL
LIN {X 0,Y 129.404,Z 581.875,A -85,B 0,C 180,E1 -25622.179,E2 -25622.179} C_VEL
LIN {X 0,Y 128.227,Z 594.991,A -85,B 0,C 180,E1 -25623.995,E2 -25623.995} C_VEL
LIN {X 0,Y 126.446,Z 608.849,A -85,B 0,C 180,E1 -25626.672,E2 -25626.672} C_VEL
LIN {X 0,Y 125.078,Z 619.84,A -85,B 0,C 180,E1 -25629.442,E2 -25629.442} C_VEL
LIN {X 0,Y 123.7,Z 631.064,A -85,B 0,C 180,E1 -25633.073,E2 -25633.073} C_VEL
LIN {X 0,Y 122.555,Z 642.084,A -85,B 0,C 180,E1 -25637.586,E2 -25637.586} C_VEL
LIN {X 0,Y 122.14,Z 651.636,A -85,B 0,C 180,E1 -25642.562,E2 -25642.562} C_VEL
LIN {X 0,Y 122.287,Z 659.233,A -85,B 0,C 180,E1 -25647.531,E2 -25647.531} C_VEL
LIN {X 0,Y 122.428,Z 664.151,A -85,B 0,C 180,E1 -25651.646,E2 -25651.646} C_VEL
LIN {X 0,Y 121.593,Z 668.355,A -85,B 0,C 180,E1 -25656.639,E2 -25656.639} C_VEL
LIN {X 0,Y 121.471,Z 672.449,A -85,B 0,C 180,E1 -25663.383,E2 -25663.383} C_VEL
LIN {X 0,Y 123.325,Z 675.139,A -85,B 0,C 180,E1 -25669.996,E2 -25669.996} C_VEL
LIN {X 0,Y 127.17,Z 676.566,A -85,B 0,C 180,E1 -25676.24,E2 -25676.24} C_VEL
LIN {X 0,Y 132.606,Z 676.73,A -85,B 0,C 180,E1 -25682.006,E2 -25682.006} C_VEL
LIN {X 0,Y 139.671,Z 675.697,A -85,B 0,C 180,E1 -25687.145,E2 -25687.145} C_VEL
LIN {X 0,Y 148.077,Z 673.442,A -85,B 0,C 180,E1 -25691.643,E2 -25691.643} C_VEL
LIN {X 0,Y 157.682,Z 669.899,A -85,B 0,C 180,E1 -25695.492,E2 -25695.492} C_VEL
LIN {X 0,Y 168.155,Z 664.955,A -85,B 0,C 180,E1 -25698.792,E2 -25698.792} C_VEL
LIN {X 0,Y 179.435,Z 658.441,A -85,B 0,C 180,E1 -25701.569,E2 -25701.569} C_VEL
LIN {X 0,Y 189.135,Z 651.769,A -85,B 0,C 180,E1 -25703.52,E2 -25703.52} C_VEL
LIN {X 0,Y 192.396,Z 649.272,A -85,B 0,C 180,E1 -25704.19,E2 -25704.19} C_VEL
LIN {X 0,Y 193.344,Z 648.517,A -85,B 0,C 180,E1 -25704.437,E2 -25704.437} C_VEL
LIN {X 0,Y 184.576,Z 654.161,A -85,B 0,C 180,E1 -25706.357,E2 -25706.357} C_VEL
LIN {X 0,Y 182.82,Z 655.151,A -85,B 0,C 180,E1 -25706.774,E2 -25706.774} C_VEL
LIN {X 0,Y 178.215,Z 657.671,A -85,B 0,C 180,E1 -25707.661,E2 -25707.661} C_VEL
LIN {X 0,Y 166.298,Z 663.003,A -85,B 0,C 180,E1 -25709.227,E2 -25709.227} C_VEL
LIN {X 0,Y 159.623,Z 665.278,A -85,B 0,C 180,E1 -25710.441,E2 -25710.441} C_VEL
LIN {X 0,Y 156.635,Z 666.045,A -85,B 0,C 180,E1 -25711.305,E2 -25711.305} C_VEL
LIN {X 0,Y 147.606,Z 667.824,A -85,B 0,C 180,E1 -25714.779,E2 -25714.779} C_VEL
LIN {X 0,Y 138.502,Z 668.436,A -85,B 0,C 180,E1 -25719.194,E2 -25719.194} C_VEL
LIN {X 0,Y 130.401,Z 667.568,A -85,B 0,C 180,E1 -25724.367,E2 -25724.367} C_VEL
LIN {X 0,Y 123.661,Z 665.258,A -85,B 0,C 180,E1 -25730.183,E2 -25730.183} C_VEL
LIN {X 0,Y 118.54,Z 661.494,A -85,B 0,C 180,E1 -25736.601,E2 -25736.601} C_VEL
LIN {X 0,Y 115.082,Z 656.04,A -85,B 0,C 180,E1 -25743.501,E2 -25743.501} C_VEL
LIN {X 0,Y 113.577,Z 650.497,A -85,B 0,C 180,E1 -25749.175,E2 -25749.175} C_VEL
LIN {X 0,Y 113.05,Z 644.326,A -85,B 0,C 180,E1 -25754.399,E2 -25754.399} C_VEL
LIN {X 0,Y 113.293,Z 636.502,A -85,B 0,C 180,E1 -25759.838,E2 -25759.838} C_VEL
LIN {X 0,Y 114,Z 628.157,A -85,B 0,C 180,E1 -25764.59,E2 -25764.59} C_VEL
LIN {X 0,Y 115.182,Z 618.183,A -85,B 0,C 180,E1 -25769.218,E2 -25769.218} C_VEL
LIN {X 0,Y 116.634,Z 607.079,A -85,B 0,C 180,E1 -25773.356,E2 -25773.356} C_VEL
LIN {X 0,Y 118.357,Z 594.742,A -85,B 0,C 180,E1 -25776.957,E2 -25776.957} C_VEL
LIN {X 0,Y 120.05,Z 582.153,A -85,B 0,C 180,E1 -25779.815,E2 -25779.815} C_VEL
LIN {X 0,Y 121.59,Z 568.139,A -85,B 0,C 180,E1 -25782.176,E2 -25782.176} C_VEL
LIN {X 0,Y 122.865,Z 553.275,A -85,B 0,C 180,E1 -25783.913,E2 -25783.913} C_VEL
LIN {X 0,Y 126.264,Z 505.395,A -85,B 0,C 180,E1 -25788.358,E2 -25788.358} C_VEL
LIN {X 0,Y 124.85,Z 500.21,A -85,B 0,C 180,E1 -25788.992,E2 -25788.992} C_VEL
LIN {X 0,Y 114.884,Z 469.168,A -85,B 0,C 180,E1 -25793.346,E2 -25793.346} C_VEL
LIN {X 0,Y 114.858,Z 469.175,A -85,B 0,C 180,E1 -25800.69,E2 -25800.69} C_VEL
LIN {X 0,Y 114.948,Z 469.167,A -85,B 0,C 180,E1 -25806.507,E2 -25806.507} C_VEL
LIN {X 0,Y 115.012,Z 469.151,A -85,B 0,C 180,E1 -25812.208,E2 -25812.208} C_VEL
LIN {X 0,Y 115.249,Z 469.128,A -85,B 0,C 180,E1 -25817.342,E2 -25817.342} C_VEL
LIN {X 0,Y 115.357,Z 469.115,A -85,B 0,C 180,E1 -25823,E2 -25823} C_VEL
LIN {X 0,Y 115.99,Z 469.03,A -85,B 0,C 180,E1 -25829.999,E2 -25829.999} C_VEL
LIN {X 0,Y 115.362,Z 469.108,A -85,B 0,C 180,E1 -25836.997,E2 -25836.997} C_VEL
LIN {X 0,Y 115.255,Z 469.128,A -85,B 0,C 180,E1 -25842.671,E2 -25842.671} C_VEL
LIN {X 0,Y 114.998,Z 469.155,A -85,B 0,C 180,E1 -25847.791,E2 -25847.791} C_VEL
LIN {X 0,Y 114.945,Z 469.163,A -85,B 0,C 180,E1 -25853.49,E2 -25853.49} C_VEL
LIN {X 0,Y 114.854,Z 469.177,A -85,B 0,C 180,E1 -25861.055,E2 -25861.055} C_VEL
LIN {X 0,Y 114.773,Z 469.188,A -85,B 0,C 180,E1 -25867.757,E2 -25867.757} C_VEL
LIN {X 0,Y 114.776,Z 469.181,A -85,B 0,C 180,E1 -25872.711,E2 -25872.711} C_VEL
LIN {X 0,Y 114.785,Z 469.186,A -85,B 0,C 180,E1 -25877.662,E2 -25877.662} C_VEL
LIN {X 0,Y 114.794,Z 469.181,A -85,B 0,C 180,E1 -25882.738,E2 -25882.738} C_VEL
LIN {X 0,Y 114.861,Z 469.172,A -85,B 0,C 180,E1 -25888.937,E2 -25888.937} C_VEL
LIN {X 0,Y 114.947,Z 469.165,A -85,B 0,C 180,E1 -25896.506,E2 -25896.506} C_VEL
LIN {X 0,Y 115.018,Z 469.157,A -85,B 0,C 180,E1 -25902.211,E2 -25902.211} C_VEL
LIN {X 0,Y 115.283,Z 469.116,A -85,B 0,C 180,E1 -25907.262,E2 -25907.262} C_VEL
LIN {X 0,Y 115.387,Z 469.111,A -85,B 0,C 180,E1 -25913.003,E2 -25913.003} C_VEL
LIN {X 0,Y 115.994,Z 469.035,A -85,B 0,C 180,E1 -25920,E2 -25920} C_VEL
LIN {X 0,Y 115.395,Z 469.108,A -85,B 0,C 180,E1 -25926.997,E2 -25926.997} C_VEL
LIN {X 0,Y 115.391,Z 469.111,A -85,B 0,C 180,E1 -25930.528,E2 -25930.528} C_VEL
LIN {X 0,Y 115.145,Z 469.134,A -85,B 0,C 180,E1 -25934.132,E2 -25934.132} C_VEL
LIN {X 0,Y 114.978,Z 469.157,A -85,B 0,C 180,E1 -25941.515,E2 -25941.515} C_VEL
LIN {X 0,Y 114.872,Z 469.175,A -85,B 0,C 180,E1 -25945.358,E2 -25945.358} C_VEL
LIN {X 0,Y 114.867,Z 469.169,A -85,B 0,C 180,E1 -25951.069,E2 -25951.069} C_VEL
LIN {X 0,Y 114.788,Z 469.184,A -85,B 0,C 180,E1 -25957.754,E2 -25957.754} C_VEL
LIN {X 0,Y 114.795,Z 469.184,A -85,B 0,C 180,E1 -25962.723,E2 -25962.723} C_VEL
LIN {X 0,Y 115.056,Z 469.246,A -85,B 0,C 180,E1 -25969.235,E2 -25969.235} C_VEL
LIN {X 0,Y 115.246,Z 470.089,A -85,B 0,C 180,E1 -25969.771,E2 -25969.771} C_VEL
LIN {X 0,Y 122.808,Z 499.874,A -85,B 0,C 180,E1 -25973.717,E2 -25973.717} C_VEL
LIN {X 0,Y 124.808,Z 537.003,A -85,B 0,C 180,E1 -25977.542,E2 -25977.542} C_VEL
LIN {X 0,Y 124.986,Z 542.532,A -85,B 0,C 180,E1 -25978.094,E2 -25978.094} C_VEL
LIN {X 0,Y 122.397,Z 580.794,A -85,B 0,C 180,E1 -25981.843,E2 -25981.843} C_VEL
LIN {X 0,Y 121.068,Z 595.064,A -85,B 0,C 180,E1 -25983.961,E2 -25983.961} C_VEL
LIN {X 0,Y 119.43,Z 607.763,A -85,B 0,C 180,E1 -25986.597,E2 -25986.597} C_VEL
LIN {X 0,Y 117.898,Z 620.141,A -85,B 0,C 180,E1 -25989.956,E2 -25989.956} C_VEL
LIN {X 0,Y 116.521,Z 631.491,A -85,B 0,C 180,E1 -25993.938,E2 -25993.938} C_VEL
LIN {X 0,Y 115.569,Z 642.033,A -85,B 0,C 180,E1 -25998.606,E2 -25998.606} C_VEL
LIN {X 0,Y 115.263,Z 651.448,A -85,B 0,C 180,E1 -26003.876,E2 -26003.876} C_VEL
LIN {X 0,Y 115.52,Z 657.739,A -85,B 0,C 180,E1 -26008.258,E2 -26008.258} C_VEL
LIN {X 0,Y 115.674,Z 661.826,A -85,B 0,C 180,E1 -26011.742,E2 -26011.742} C_VEL
LIN {X 0,Y 115.044,Z 664.923,A -85,B 0,C 180,E1 -26015.259,E2 -26015.259} C_VEL
LIN {X 0,Y 114.557,Z 668.958,A -85,B 0,C 180,E1 -26021.009,E2 -26021.009} C_VEL
LIN {X 0,Y 115.532,Z 672.352,A -85,B 0,C 180,E1 -26027.709,E2 -26027.709} C_VEL
LIN {X 0,Y 118.566,Z 674.72,A -85,B 0,C 180,E1 -26034.516,E2 -26034.516} C_VEL
LIN {X 0,Y 123.547,Z 675.856,A -85,B 0,C 180,E1 -26040.796,E2 -26040.796} C_VEL
LIN {X 0,Y 130.2,Z 675.811,A -85,B 0,C 180,E1 -26046.426,E2 -26046.426} C_VEL
LIN {X 0,Y 138.329,Z 674.576,A -85,B 0,C 180,E1 -26051.338,E2 -26051.338} C_VEL
LIN {X 0,Y 147.681,Z 672.138,A -85,B 0,C 180,E1 -26055.55,E2 -26055.55} C_VEL
LIN {X 0,Y 158.12,Z 668.37,A -85,B 0,C 180,E1 -26059.08,E2 -26059.08} C_VEL
LIN {X 0,Y 169.328,Z 663.233,A -85,B 0,C 180,E1 -26062.056,E2 -26062.056} C_VEL
LIN {X 0,Y 179.09,Z 657.778,A -85,B 0,C 180,E1 -26064.15,E2 -26064.15} C_VEL
LIN {X 0,Y 180.245,Z 657.006,A -85,B 0,C 180,E1 -26064.761,E2 -26064.761} C_VEL
LIN {X 0,Y 169.482,Z 661.919,A -85,B 0,C 180,E1 -26067.379,E2 -26067.379} C_VEL
LIN {X 0,Y 163.754,Z 664.004,A -85,B 0,C 180,E1 -26069.001,E2 -26069.001} C_VEL
LIN {X 0,Y 156.635,Z 666.045,A -85,B 0,C 180,E1 -26071.305,E2 -26071.305} C_VEL
LIN {X 0,Y 152.033,Z 667.158,A -85,B 0,C 180,E1 -26072.636,E2 -26072.636} C_VEL
LIN {X 0,Y 143.466,Z 668.556,A -85,B 0,C 180,E1 -26074.505,E2 -26074.505} C_VEL
LIN {X 0,Y 136.702,Z 669.126,A -85,B 0,C 180,E1 -26076.159,E2 -26076.159} C_VEL
LIN {X 0,Y 132.248,Z 669.073,A -85,B 0,C 180,E1 -26077.789,E2 -26077.789} C_VEL
LIN {X 0,Y 130.99,Z 668.951,A -85,B 0,C 180,E1 -26078.439,E2 -26078.439} C_VEL
LIN {X 0,Y 123.349,Z 667.546,A -85,B 0,C 180,E1 -26083.448,E2 -26083.448} C_VEL
LIN {X 0,Y 116.48,Z 664.641,A -85,B 0,C 180,E1 -26089.571,E2 -26089.571} C_VEL
LIN {X 0,Y 111.277,Z 660.246,A -85,B 0,C 180,E1 -26096.379,E2 -26096.379} C_VEL
LIN {X 0,Y 108.531,Z 655.895,A -85,B 0,C 180,E1 -26101.855,E2 -26101.855} C_VEL
LIN {X 0,Y 106.65,Z 649.241,A -85,B 0,C 180,E1 -26108.701,E2 -26108.701} C_VEL
LIN {X 0,Y 106.099,Z 641.31,A -85,B 0,C 180,E1 -26115.364,E2 -26115.364} C_VEL
LIN {X 0,Y 106.467,Z 632.962,A -85,B 0,C 180,E1 -26121.048,E2 -26121.048} C_VEL
LIN {X 0,Y 107.39,Z 623.508,A -85,B 0,C 180,E1 -26126.215,E2 -26126.215} C_VEL
LIN {X 0,Y 108.769,Z 612.372,A -85,B 0,C 180,E1 -26131.125,E2 -26131.125} C_VEL
LIN {X 0,Y 110.522,Z 599.83,A -85,B 0,C 180,E1 -26135.468,E2 -26135.468} C_VEL
LIN {X 0,Y 112.337,Z 586.578,A -85,B 0,C 180,E1 -26139.015,E2 -26139.015} C_VEL
LIN {X 0,Y 113.896,Z 573.847,A -85,B 0,C 180,E1 -26141.554,E2 -26141.554} C_VEL
LIN {X 0,Y 115.226,Z 560.086,A -85,B 0,C 180,E1 -26143.551,E2 -26143.551} C_VEL
LIN {X 0,Y 119.172,Z 505.531,A -85,B 0,C 180,E1 -26148.997,E2 -26148.997} C_VEL
LIN {X 0,Y 107.874,Z 470.04,A -85,B 0,C 180,E1 -26154.323,E2 -26154.323} C_VEL
LIN {X 0,Y 107.796,Z 470.058,A -85,B 0,C 180,E1 -26158.56,E2 -26158.56} C_VEL
LIN {X 0,Y 107.912,Z 470.043,A -85,B 0,C 180,E1 -26166.996,E2 -26166.996} C_VEL
LIN {X 0,Y 108.031,Z 470.028,A -85,B 0,C 180,E1 -26174.915,E2 -26174.915} C_VEL
LIN {X 0,Y 108.25,Z 469.996,A -85,B 0,C 180,E1 -26178.767,E2 -26178.767} C_VEL
LIN {X 0,Y 108.438,Z 469.976,A -85,B 0,C 180,E1 -26186.283,E2 -26186.283} C_VEL
LIN {X 0,Y 108.915,Z 469.911,A -85,B 0,C 180,E1 -26189.999,E2 -26189.999} C_VEL
LIN {X 0,Y 108.302,Z 469.987,A -85,B 0,C 180,E1 -26197.456,E2 -26197.456} C_VEL
LIN {X 0,Y 108.175,Z 470.01,A -85,B 0,C 180,E1 -26202.959,E2 -26202.959} C_VEL
LIN {X 0,Y 107.894,Z 470.044,A -85,B 0,C 180,E1 -26209.006,E2 -26209.006} C_VEL
LIN {X 0,Y 107.854,Z 470.044,A -85,B 0,C 180,E1 -26214.18,E2 -26214.18} C_VEL
LIN {X 0,Y 107.777,Z 470.057,A -85,B 0,C 180,E1 -26222.037,E2 -26222.037} C_VEL
LIN {X 0,Y 107.682,Z 470.073,A -85,B 0,C 180,E1 -26228.446,E2 -26228.446} C_VEL
LIN {X 0,Y 107.668,Z 470.072,A -85,B 0,C 180,E1 -26235.89,E2 -26235.89} C_VEL
LIN {X 0,Y 107.689,Z 470.062,A -85,B 0,C 180,E1 -26241.547,E2 -26241.547} C_VEL
LIN {X 0,Y 107.799,Z 470.052,A -85,B 0,C 180,E1 -26248.563,E2 -26248.563} C_VEL
LIN {X 0,Y 107.911,Z 470.039,A -85,B 0,C 180,E1 -26256.998,E2 -26256.998} C_VEL
LIN {X 0,Y 108.039,Z 470.025,A -85,B 0,C 180,E1 -26264.918,E2 -26264.918} C_VEL
LIN {X 0,Y 108.287,Z 469.99,A -85,B 0,C 180,E1 -26268.773,E2 -26268.773} C_VEL
LIN {X 0,Y 108.455,Z 469.968,A -85,B 0,C 180,E1 -26276.285,E2 -26276.285} C_VEL
LIN {X 0,Y 108.944,Z 469.914,A -85,B 0,C 180,E1 -26280,E2 -26280} C_VEL
LIN {X 0,Y 108.338,Z 469.988,A -85,B 0,C 180,E1 -26287.455,E2 -26287.455} C_VEL
LIN {X 0,Y 108.202,Z 469.999,A -85,B 0,C 180,E1 -26293.026,E2 -26293.026} C_VEL
LIN {X 0,Y 107.904,Z 470.043,A -85,B 0,C 180,E1 -26299.006,E2 -26299.006} C_VEL
LIN {X 0,Y 107.857,Z 470.045,A -85,B 0,C 180,E1 -26304.185,E2 -26304.185} C_VEL
LIN {X 0,Y 107.791,Z 470.051,A -85,B 0,C 180,E1 -26312.051,E2 -26312.051} C_VEL
LIN {X 0,Y 107.695,Z 470.065,A -85,B 0,C 180,E1 -26318.457,E2 -26318.457} C_VEL
LIN {X 0,Y 107.758,Z 470.061,A -85,B 0,C 180,E1 -26325.843,E2 -26325.843} C_VEL
LIN {X 0,Y 107.941,Z 470.032,A -85,B 0,C 180,E1 -26328.683,E2 -26328.683} C_VEL
LIN {X 0,Y 113.442,Z 491.193,A -85,B 0,C 180,E1 -26331.825,E2 -26331.825} C_VEL
LIN {X 0,Y 115.856,Z 501.222,A -85,B 0,C 180,E1 -26333.164,E2 -26333.164} C_VEL
LIN {X 0,Y 117.938,Z 542.803,A -85,B 0,C 180,E1 -26337.695,E2 -26337.695} C_VEL
LIN {X 0,Y 115.291,Z 580.707,A -85,B 0,C 180,E1 -26341.685,E2 -26341.685} C_VEL
LIN {X 0,Y 113.963,Z 594.82,A -85,B 0,C 180,E1 -26343.936,E2 -26343.936} C_VEL
LIN {X 0,Y 112.22,Z 608.308,A -85,B 0,C 180,E1 -26346.959,E2 -26346.959} C_VEL
LIN {X 0,Y 110.725,Z 620.398,A -85,B 0,C 180,E1 -26350.536,E2 -26350.536} C_VEL
LIN {X 0,Y 109.385,Z 631.658,A -85,B 0,C 180,E1 -26354.81,E2 -26354.81} C_VEL
LIN {X 0,Y 108.716,Z 640.147,A -85,B 0,C 180,E1 -26358.819,E2 -26358.819} C_VEL
LIN {X 0,Y 108.479,Z 648.292,A -85,B 0,C 180,E1 -26363.491,E2 -26363.491} C_VEL
LIN {X 0,Y 108.72,Z 654.976,A -85,B 0,C 180,E1 -26368.149,E2 -26368.149} C_VEL
LIN {X 0,Y 108.946,Z 659.32,A -85,B 0,C 180,E1 -26371.85,E2 -26371.85} C_VEL
LIN {X 0,Y 108.739,Z 661.132,A -85,B 0,C 180,E1 -26373.707,E2 -26373.707} C_VEL
LIN {X 0,Y 107.942,Z 665.451,A -85,B 0,C 180,E1 -26379.369,E2 -26379.369} C_VEL
LIN {X 0,Y 108.123,Z 668.799,A -85,B 0,C 180,E1 -26385.071,E2 -26385.071} C_VEL
LIN {X 0,Y 110.308,Z 672.133,A -85,B 0,C 180,E1 -26392.476,E2 -26392.476} C_VEL
LIN {X 0,Y 114.693,Z 674.229,A -85,B 0,C 180,E1 -26399.356,E2 -26399.356} C_VEL
LIN {X 0,Y 120.859,Z 675.127,A -85,B 0,C 180,E1 -26405.558,E2 -26405.558} C_VEL
LIN {X 0,Y 128.677,Z 674.874,A -85,B 0,C 180,E1 -26410.952,E2 -26410.952} C_VEL
LIN {X 0,Y 137.796,Z 673.444,A -85,B 0,C 180,E1 -26415.566,E2 -26415.566} C_VEL
LIN {X 0,Y 148.101,Z 670.795,A -85,B 0,C 180,E1 -26419.401,E2 -26419.401} C_VEL
LIN {X 0,Y 159.228,Z 666.895,A -85,B 0,C 180,E1 -26422.608,E2 -26422.608} C_VEL
LIN {X 0,Y 166.362,Z 663.838,A -85,B 0,C 180,E1 -26424.257,E2 -26424.257} C_VEL
LIN {X 0,Y 167.16,Z 663.344,A -85,B 0,C 180,E1 -26425.075,E2 -26425.075} C_VEL
LIN {X 0,Y 157.609,Z 666.307,A -85,B 0,C 180,E1 -26427.649,E2 -26427.649} C_VEL
LIN {X 0,Y 146.485,Z 668.497,A -85,B 0,C 180,E1 -26431.329,E2 -26431.329} C_VEL
LIN {X 0,Y 136.319,Z 669.217,A -85,B 0,C 180,E1 -26435.641,E2 -26435.641} C_VEL
LIN {X 0,Y 130.99,Z 668.951,A -85,B 0,C 180,E1 -26438.439,E2 -26438.439} C_VEL
LIN {X 0,Y 127.006,Z 668.54,A -85,B 0,C 180,E1 -26440.362,E2 -26440.362} C_VEL
LIN {X 0,Y 119.436,Z 667.309,A -85,B 0,C 180,E1 -26443.281,E2 -26443.281} C_VEL
LIN {X 0,Y 112.338,Z 665.267,A -85,B 0,C 180,E1 -26446.547,E2 -26446.547} C_VEL
LIN {X 0,Y 109.212,Z 663.659,A -85,B 0,C 180,E1 -26449,E2 -26449} C_VEL
LIN {X 0,Y 105.195,Z 660.114,A -85,B 0,C 180,E1 -26454.246,E2 -26454.246} C_VEL
LIN {X 0,Y 101.353,Z 653.857,A -85,B 0,C 180,E1 -26461.987,E2 -26461.987} C_VEL
LIN {X 0,Y 99.614,Z 646.984,A -85,B 0,C 180,E1 -26468.974,E2 -26468.974} C_VEL
LIN {X 0,Y 99.204,Z 639.285,A -85,B 0,C 180,E1 -26475.406,E2 -26475.406} C_VEL
LIN {X 0,Y 99.538,Z 631.719,A -85,B 0,C 180,E1 -26480.673,E2 -26480.673} C_VEL
LIN {X 0,Y 100.482,Z 621.555,A -85,B 0,C 180,E1 -26486.48,E2 -26486.48} C_VEL
LIN {X 0,Y 101.774,Z 611.112,A -85,B 0,C 180,E1 -26491.192,E2 -26491.192} C_VEL
LIN {X 0,Y 103.602,Z 598.123,A -85,B 0,C 180,E1 -26495.834,E2 -26495.834} C_VEL
LIN {X 0,Y 105.515,Z 584.319,A -85,B 0,C 180,E1 -26499.563,E2 -26499.563} C_VEL
LIN {X 0,Y 107.111,Z 570.854,A -85,B 0,C 180,E1 -26502.267,E2 -26502.267} C_VEL
LIN {X 0,Y 108.495,Z 556.563,A -85,B 0,C 180,E1 -26504.283,E2 -26504.283} C_VEL
LIN {X 0,Y 112.139,Z 506.565,A -85,B 0,C 180,E1 -26509.616,E2 -26509.616} C_VEL
LIN {X 0,Y 100.78,Z 470.926,A -85,B 0,C 180,E1 -26515.257,E2 -26515.257} C_VEL
LIN {X 0,Y 100.654,Z 470.944,A -85,B 0,C 180,E1 -26520.739,E2 -26520.739} C_VEL
LIN {X 0,Y 100.788,Z 470.929,A -85,B 0,C 180,E1 -26525.266,E2 -26525.266} C_VEL
LIN {X 0,Y 100.817,Z 470.924,A -85,B 0,C 180,E1 -26529.6,E2 -26529.6} C_VEL
LIN {X 0,Y 101.1,Z 470.891,A -85,B 0,C 180,E1 -26536.708,E2 -26536.708} C_VEL
LIN {X 0,Y 101.237,Z 470.87,A -85,B 0,C 180,E1 -26542.018,E2 -26542.018} C_VEL
LIN {X 0,Y 101.843,Z 470.792,A -85,B 0,C 180,E1 -26549.999,E2 -26549.999} C_VEL
LIN {X 0,Y 101.241,Z 470.866,A -85,B 0,C 180,E1 -26557.979,E2 -26557.979} C_VEL
LIN {X 0,Y 101.104,Z 470.89,A -85,B 0,C 180,E1 -26563.3,E2 -26563.3} C_VEL
LIN {X 0,Y 100.809,Z 470.928,A -85,B 0,C 180,E1 -26570.399,E2 -26570.399} C_VEL
LIN {X 0,Y 100.774,Z 470.924,A -85,B 0,C 180,E1 -26574.957,E2 -26574.957} C_VEL
LIN {X 0,Y 100.686,Z 470.936,A -85,B 0,C 180,E1 -26583.111,E2 -26583.111} C_VEL
LIN {X 0,Y 100.633,Z 470.949,A -85,B 0,C 180,E1 -26589.806,E2 -26589.806} C_VEL
LIN {X 0,Y 100.639,Z 470.948,A -85,B 0,C 180,E1 -26595.706,E2 -26595.706} C_VEL
LIN {X 0,Y 100.626,Z 470.942,A -85,B 0,C 180,E1 -26601.055,E2 -26601.055} C_VEL
LIN {X 0,Y 100.693,Z 470.941,A -85,B 0,C 180,E1 -26606.881,E2 -26606.881} C_VEL
LIN {X 0,Y 100.784,Z 470.93,A -85,B 0,C 180,E1 -26615.267,E2 -26615.267} C_VEL
LIN {X 0,Y 100.818,Z 470.92,A -85,B 0,C 180,E1 -26619.602,E2 -26619.602} C_VEL
LIN {X 0,Y 101.186,Z 470.872,A -85,B 0,C 180,E1 -26627.974,E2 -26627.974} C_VEL
LIN {X 0,Y 101.266,Z 470.871,A -85,B 0,C 180,E1 -26632.022,E2 -26632.022} C_VEL
LIN {X 0,Y 101.868,Z 470.795,A -85,B 0,C 180,E1 -26640,E2 -26640} C_VEL
LIN {X 0,Y 101.277,Z 470.868,A -85,B 0,C 180,E1 -26647.978,E2 -26647.978} C_VEL
LIN {X 0,Y 101.113,Z 470.882,A -85,B 0,C 180,E1 -26653.327,E2 -26653.327} C_VEL
LIN {X 0,Y 100.815,Z 470.924,A -85,B 0,C 180,E1 -26660.4,E2 -26660.4} C_VEL
LIN {X 0,Y 100.773,Z 470.93,A -85,B 0,C 180,E1 -26664.959,E2 -26664.959} C_VEL
LIN {X 0,Y 100.696,Z 470.938,A -85,B 0,C 180,E1 -26673.122,E2 -26673.122} C_VEL
LIN {X 0,Y 100.646,Z 470.94,A -85,B 0,C 180,E1 -26679.817,E2 -26679.817} C_VEL
LIN {X 0,Y 100.833,Z 470.919,A -85,B 0,C 180,E1 -26687.648,E2 -26687.648} C_VEL
LIN {X 0,Y 104.038,Z 482.194,A -85,B 0,C 180,E1 -26689.567,E2 -26689.567} C_VEL
LIN {X 0,Y 108.935,Z 502.574,A -85,B 0,C 180,E1 -26692.558,E2 -26692.558} C_VEL
LIN {X 0,Y 110.948,Z 542.011,A -85,B 0,C 180,E1 -26697.162,E2 -26697.162} C_VEL
LIN {X 0,Y 108.199,Z 580.632,A -85,B 0,C 180,E1 -26701.511,E2 -26701.511} C_VEL
LIN {X 0,Y 106.878,Z 594.592,A -85,B 0,C 180,E1 -26703.913,E2 -26703.913} C_VEL
LIN {X 0,Y 105.241,Z 607.059,A -85,B 0,C 180,E1 -26706.902,E2 -26706.902} C_VEL
LIN {X 0,Y 103.755,Z 619.242,A -85,B 0,C 180,E1 -26710.74,E2 -26710.74} C_VEL
LIN {X 0,Y 102.477,Z 630.294,A -85,B 0,C 180,E1 -26715.232,E2 -26715.232} C_VEL
LIN {X 0,Y 101.786,Z 639.858,A -85,B 0,C 180,E1 -26720.061,E2 -26720.061} C_VEL
LIN {X 0,Y 101.693,Z 647.904,A -85,B 0,C 180,E1 -26725.046,E2 -26725.046} C_VEL
LIN {X 0,Y 102.118,Z 654.519,A -85,B 0,C 180,E1 -26730.001,E2 -26730.001} C_VEL
LIN {X 0,Y 102.258,Z 656.733,A -85,B 0,C 180,E1 -26731.971,E2 -26731.971} C_VEL
LIN {X 0,Y 102.098,Z 658.61,A -85,B 0,C 180,E1 -26733.949,E2 -26733.949} C_VEL
LIN {X 0,Y 101.313,Z 663.179,A -85,B 0,C 180,E1 -26739.988,E2 -26739.988} C_VEL
LIN {X 0,Y 101.548,Z 666.828,A -85,B 0,C 180,E1 -26746.073,E2 -26746.073} C_VEL
LIN {X 0,Y 103.946,Z 670.447,A -85,B 0,C 180,E1 -26753.935,E2 -26753.935} C_VEL
LIN {X 0,Y 108.639,Z 672.873,A -85,B 0,C 180,E1 -26761.168,E2 -26761.168} C_VEL
LIN {X 0,Y 115.209,Z 674.111,A -85,B 0,C 180,E1 -26767.593,E2 -26767.593} C_VEL
LIN {X 0,Y 123.43,Z 674.234,A -85,B 0,C 180,E1 -26773.102,E2 -26773.102} C_VEL
LIN {X 0,Y 132.934,Z 673.218,A -85,B 0,C 180,E1 -26777.747,E2 -26777.747} C_VEL
LIN {X 0,Y 143.599,Z 671.049,A -85,B 0,C 180,E1 -26781.544,E2 -26781.544} C_VEL
LIN {X 0,Y 155.046,Z 667.637,A -85,B 0,C 180,E1 -26784.679,E2 -26784.679} C_VEL
LIN {X 0,Y 153.125,Z 667.961,A -85,B 0,C 180,E1 -26785.707,E2 -26785.707} C_VEL
LIN {X 0,Y 145.689,Z 669.229,A -85,B 0,C 180,E1 -26787.951,E2 -26787.951} C_VEL
LIN {X 0,Y 134.737,Z 670.004,A -85,B 0,C 180,E1 -26792.001,E2 -26792.001} C_VEL
LIN {X 0,Y 124.89,Z 669.357,A -85,B 0,C 180,E1 -26796.801,E2 -26796.801} C_VEL
LIN {X 0,Y 116.339,Z 667.251,A -85,B 0,C 180,E1 -26802.419,E2 -26802.419} C_VEL
LIN {X 0,Y 109.212,Z 663.659,A -85,B 0,C 180,E1 -26809,E2 -26809} C_VEL
LIN {X 0,Y 106.361,Z 661.865,A -85,B 0,C 180,E1 -26811.564,E2 -26811.564} C_VEL
LIN {X 0,Y 100.69,Z 658.159,A -85,B 0,C 180,E1 -26815.572,E2 -26815.572} C_VEL
LIN {X 0,Y 95.687,Z 653.745,A -85,B 0,C 180,E1 -26819.884,E2 -26819.884} C_VEL
LIN {X 0,Y 93.999,Z 650.848,A -85,B 0,C 180,E1 -26822.841,E2 -26822.841} C_VEL
LIN {X 0,Y 92.481,Z 642.561,A -85,B 0,C 180,E1 -26830.949,E2 -26830.949} C_VEL
LIN {X 0,Y 92.424,Z 634.083,A -85,B 0,C 180,E1 -26837.707,E2 -26837.707} C_VEL
LIN {X 0,Y 93.012,Z 625.42,A -85,B 0,C 180,E1 -26843.338,E2 -26843.338} C_VEL
LIN {X 0,Y 94.198,Z 614.685,A -85,B 0,C 180,E1 -26849.009,E2 -26849.009} C_VEL
LIN {X 0,Y 95.763,Z 602.734,A -85,B 0,C 180,E1 -26854.028,E2 -26854.028} C_VEL
LIN {X 0,Y 97.403,Z 591.253,A -85,B 0,C 180,E1 -26857.761,E2 -26857.761} C_VEL
LIN {X 0,Y 99.138,Z 578.459,A -85,B 0,C 180,E1 -26860.976,E2 -26860.976} C_VEL
LIN {X 0,Y 100.719,Z 564.264,A -85,B 0,C 180,E1 -26863.556,E2 -26863.556} C_VEL
LIN {X 0,Y 102.688,Z 539.412,A -85,B 0,C 180,E1 -26866.604,E2 -26866.604} C_VEL
LIN {X 0,Y 105.063,Z 507.69,A -85,B 0,C 180,E1 -26870.189,E2 -26870.189} C_VEL
LIN {X 0,Y 94.378,Z 474.087,A -85,B 0,C 180,E1 -26875.863,E2 -26875.863} C_VEL
LIN {X 0,Y 93.716,Z 471.808,A -85,B 0,C 180,E1 -26876.388,E2 -26876.388} C_VEL
LIN {X 0,Y 93.67,Z 471.811,A -85,B 0,C 180,E1 -26884.205,E2 -26884.205} C_VEL
LIN {X 0,Y 93.694,Z 471.814,A -85,B 0,C 180,E1 -26887.971,E2 -26887.971} C_VEL
LIN {X 0,Y 94.021,Z 471.774,A -85,B 0,C 180,E1 -26896.347,E2 -26896.347} C_VEL
LIN {X 0,Y 94.171,Z 471.749,A -85,B 0,C 180,E1 -26901.414,E2 -26901.414} C_VEL
LIN {X 0,Y 94.772,Z 471.673,A -85,B 0,C 180,E1 -26909.998,E2 -26909.998} C_VEL
LIN {X 0,Y 94.175,Z 471.747,A -85,B 0,C 180,E1 -26918.582,E2 -26918.582} C_VEL
LIN {X 0,Y 94.023,Z 471.772,A -85,B 0,C 180,E1 -26923.66,E2 -26923.66} C_VEL
LIN {X 0,Y 93.689,Z 471.815,A -85,B 0,C 180,E1 -26932.027,E2 -26932.027} C_VEL
LIN {X 0,Y 93.618,Z 471.818,A -85,B 0,C 180,E1 -26936.769,E2 -26936.769} C_VEL
LIN {X 0,Y 93.583,Z 471.82,A -85,B 0,C 180,E1 -26944.301,E2 -26944.301} C_VEL
LIN {X 0,Y 93.526,Z 471.827,A -85,B 0,C 180,E1 -26952.554,E2 -26952.554} C_VEL
LIN {X 0,Y 93.532,Z 471.832,A -85,B 0,C 180,E1 -26958.71,E2 -26958.71} C_VEL
LIN {X 0,Y 93.589,Z 471.827,A -85,B 0,C 180,E1 -26965.691,E2 -26965.691} C_VEL
LIN {X 0,Y 93.667,Z 471.817,A -85,B 0,C 180,E1 -26974.205,E2 -26974.205} C_VEL
LIN {X 0,Y 93.693,Z 471.808,A -85,B 0,C 180,E1 -26977.973,E2 -26977.973} C_VEL
LIN {X 0,Y 94.09,Z 471.756,A -85,B 0,C 180,E1 -26987.051,E2 -26987.051} C_VEL
LIN {X 0,Y 94.199,Z 471.751,A -85,B 0,C 180,E1 -26991.419,E2 -26991.419} C_VEL
LIN {X 0,Y 94.794,Z 471.676,A -85,B 0,C 180,E1 -27000,E2 -27000} C_VEL
LIN {X 0,Y 94.209,Z 471.75,A -85,B 0,C 180,E1 -27008.581,E2 -27008.581} C_VEL
LIN {X 0,Y 94.034,Z 471.763,A -85,B 0,C 180,E1 -27013.692,E2 -27013.692} C_VEL
LIN {X 0,Y 93.691,Z 471.807,A -85,B 0,C 180,E1 -27022.029,E2 -27022.029} C_VEL
LIN {X 0,Y 93.622,Z 471.824,A -85,B 0,C 180,E1 -27026.77,E2 -27026.77} C_VEL
LIN {X 0,Y 93.593,Z 471.825,A -85,B 0,C 180,E1 -27034.312,E2 -27034.312} C_VEL
LIN {X 0,Y 93.564,Z 471.828,A -85,B 0,C 180,E1 -27042.535,E2 -27042.535} C_VEL
LIN {X 0,Y 93.719,Z 471.808,A -85,B 0,C 180,E1 -27046.568,E2 -27046.568} C_VEL
LIN {X 0,Y 96.337,Z 480.374,A -85,B 0,C 180,E1 -27048.201,E2 -27048.201} C_VEL
LIN {X 0,Y 102.013,Z 503.599,A -85,B 0,C 180,E1 -27051.874,E2 -27051.874} C_VEL
LIN {X 0,Y 103.849,Z 542.844,A -85,B 0,C 180,E1 -27056.763,E2 -27056.763} C_VEL
LIN {X 0,Y 101.138,Z 580.057,A -85,B 0,C 180,E1 -27061.322,E2 -27061.322} C_VEL
LIN {X 0,Y 99.814,Z 593.879,A -85,B 0,C 180,E1 -27063.893,E2 -27063.893} C_VEL
LIN {X 0,Y 98.071,Z 607.131,A -85,B 0,C 180,E1 -27067.346,E2 -27067.346} C_VEL
LIN {X 0,Y 96.768,Z 618.26,A -85,B 0,C 180,E1 -27071.119,E2 -27071.119} C_VEL
LIN {X 0,Y 95.613,Z 628.383,A -85,B 0,C 180,E1 -27075.471,E2 -27075.471} C_VEL
LIN {X 0,Y 94.981,Z 637.744,A -85,B 0,C 180,E1 -27080.418,E2 -27080.418} C_VEL
LIN {X 0,Y 94.981,Z 646.005,A -85,B 0,C 180,E1 -27085.758,E2 -27085.758} C_VEL
LIN {X 0,Y 95.493,Z 652.699,A -85,B 0,C 180,E1 -27091.056,E2 -27091.056} C_VEL
LIN {X 0,Y 95.533,Z 655.914,A -85,B 0,C 180,E1 -27094.22,E2 -27094.22} C_VEL
LIN {X 0,Y 94.724,Z 660.776,A -85,B 0,C 180,E1 -27100.691,E2 -27100.691} C_VEL
LIN {X 0,Y 95.501,Z 665.739,A -85,B 0,C 180,E1 -27109.341,E2 -27109.341} C_VEL
LIN {X 0,Y 97.691,Z 668.603,A -85,B 0,C 180,E1 -27115.574,E2 -27115.574} C_VEL
LIN {X 0,Y 102.755,Z 671.351,A -85,B 0,C 180,E1 -27123.174,E2 -27123.174} C_VEL
LIN {X 0,Y 109.723,Z 672.958,A -85,B 0,C 180,E1 -27129.833,E2 -27129.833} C_VEL
LIN {X 0,Y 118.374,Z 673.463,A -85,B 0,C 180,E1 -27135.437,E2 -27135.437} C_VEL
LIN {X 0,Y 128.281,Z 672.867,A -85,B 0,C 180,E1 -27140.087,E2 -27140.087} C_VEL
LIN {X 0,Y 139.296,Z 671.146,A -85,B 0,C 180,E1 -27143.831,E2 -27143.831} C_VEL
LIN {X 0,Y 141.154,Z 670.781,A -85,B 0,C 180,E1 -27144.347,E2 -27144.347} C_VEL
LIN {X 0,Y 142.628,Z 670.303,A -85,B 0,C 180,E1 -27145.388,E2 -27145.388} C_VEL
LIN {X 0,Y 130.423,Z 670.779,A -85,B 0,C 180,E1 -27149.565,E2 -27149.565} C_VEL
LIN {X 0,Y 123.063,Z 670.212,A -85,B 0,C 180,E1 -27152.814,E2 -27152.814} C_VEL
LIN {X 0,Y 113.478,Z 668.164,A -85,B 0,C 180,E1 -27158.282,E2 -27158.282} C_VEL
LIN {X 0,Y 105.543,Z 664.775,A -85,B 0,C 180,E1 -27164.552,E2 -27164.552} C_VEL
LIN {X 0,Y 99.266,Z 659.918,A -85,B 0,C 180,E1 -27171.859,E2 -27171.859} C_VEL
LIN {X 0,Y 95.811,Z 655.197,A -85,B 0,C 180,E1 -27177.898,E2 -27177.898} C_VEL
LIN {X 0,Y 93.999,Z 650.848,A -85,B 0,C 180,E1 -27182.841,E2 -27182.841} C_VEL
LIN {X 0,Y 92.606,Z 647.801,A -85,B 0,C 180,E1 -27185.785,E2 -27185.785} C_VEL
LIN {X 0,Y 89.165,Z 642.057,A -85,B 0,C 180,E1 -27190.334,E2 -27190.334} C_VEL
LIN {X 0,Y 86.167,Z 635.566,A -85,B 0,C 180,E1 -27194.953,E2 -27194.953} C_VEL
LIN {X 0,Y 85.58,Z 631.487,A -85,B 0,C 180,E1 -27197.901,E2 -27197.901} C_VEL
LIN {X 0,Y 86.225,Z 622.187,A -85,B 0,C 180,E1 -27204.05,E2 -27204.05} C_VEL
LIN {X 0,Y 87.406,Z 611.957,A -85,B 0,C 180,E1 -27209.504,E2 -27209.504} C_VEL
LIN {X 0,Y 89.096,Z 599.245,A -85,B 0,C 180,E1 -27214.882,E2 -27214.882} C_VEL
LIN {X 0,Y 90.985,Z 585.97,A -85,B 0,C 180,E1 -27219.141,E2 -27219.141} C_VEL
LIN {X 0,Y 92.663,Z 572.888,A -85,B 0,C 180,E1 -27222.292,E2 -27222.292} C_VEL
LIN {X 0,Y 94.083,Z 558.994,A -85,B 0,C 180,E1 -27224.64,E2 -27224.64} C_VEL
LIN {X 0,Y 98.03,Z 508.849,A -85,B 0,C 180,E1 -27230.822,E2 -27230.822} C_VEL
LIN {X 0,Y 87.874,Z 476.664,A -85,B 0,C 180,E1 -27236.641,E2 -27236.641} C_VEL
LIN {X 0,Y 86.63,Z 472.693,A -85,B 0,C 180,E1 -27237.487,E2 -27237.487} C_VEL
LIN {X 0,Y 86.588,Z 472.698,A -85,B 0,C 180,E1 -27246.055,E2 -27246.055} C_VEL
LIN {X 0,Y 86.646,Z 472.683,A -85,B 0,C 180,E1 -27251.066,E2 -27251.066} C_VEL
LIN {X 0,Y 86.932,Z 472.656,A -85,B 0,C 180,E1 -27255.962,E2 -27255.962} C_VEL
LIN {X 0,Y 87.081,Z 472.63,A -85,B 0,C 180,E1 -27260.709,E2 -27260.709} C_VEL
LIN {X 0,Y 87.701,Z 472.553,A -85,B 0,C 180,E1 -27269.998,E2 -27269.998} C_VEL
LIN {X 0,Y 87.084,Z 472.632,A -85,B 0,C 180,E1 -27279.287,E2 -27279.287} C_VEL
LIN {X 0,Y 86.931,Z 472.654,A -85,B 0,C 180,E1 -27284.035,E2 -27284.035} C_VEL
LIN {X 0,Y 86.641,Z 472.69,A -85,B 0,C 180,E1 -27288.931,E2 -27288.931} C_VEL
LIN {X 0,Y 86.582,Z 472.694,A -85,B 0,C 180,E1 -27296.761,E2 -27296.761} C_VEL
LIN {X 0,Y 86.501,Z 472.706,A -85,B 0,C 180,E1 -27305.662,E2 -27305.662} C_VEL
LIN {X 0,Y 86.47,Z 472.706,A -85,B 0,C 180,E1 -27312.989,E2 -27312.989} C_VEL
LIN {X 0,Y 86.454,Z 472.713,A -85,B 0,C 180,E1 -27319.434,E2 -27319.434} C_VEL
LIN {X 0,Y 86.532,Z 472.706,A -85,B 0,C 180,E1 -27325.353,E2 -27325.353} C_VEL
LIN {X 0,Y 86.582,Z 472.7,A -85,B 0,C 180,E1 -27333.235,E2 -27333.235} C_VEL
LIN {X 0,Y 86.647,Z 472.689,A -85,B 0,C 180,E1 -27341.069,E2 -27341.069} C_VEL
LIN {X 0,Y 86.968,Z 472.647,A -85,B 0,C 180,E1 -27345.97,E2 -27345.97} C_VEL
LIN {X 0,Y 87.107,Z 472.634,A -85,B 0,C 180,E1 -27350.714,E2 -27350.714} C_VEL
LIN {X 0,Y 87.722,Z 472.557,A -85,B 0,C 180,E1 -27360,E2 -27360} C_VEL
LIN {X 0,Y 87.113,Z 472.634,A -85,B 0,C 180,E1 -27369.286,E2 -27369.286} C_VEL
LIN {X 0,Y 86.949,Z 472.645,A -85,B 0,C 180,E1 -27374.088,E2 -27374.088} C_VEL
LIN {X 0,Y 86.661,Z 472.69,A -85,B 0,C 180,E1 -27378.929,E2 -27378.929} C_VEL
LIN {X 0,Y 86.584,Z 472.701,A -85,B 0,C 180,E1 -27386.768,E2 -27386.768} C_VEL
LIN {X 0,Y 86.511,Z 472.709,A -85,B 0,C 180,E1 -27395.673,E2 -27395.673} C_VEL
LIN {X 0,Y 86.589,Z 472.7,A -85,B 0,C 180,E1 -27404.727,E2 -27404.727} C_VEL
LIN {X 0,Y 86.624,Z 472.694,A -85,B 0,C 180,E1 -27405.382,E2 -27405.382} C_VEL
LIN {X 0,Y 89.954,Z 483.366,A -85,B 0,C 180,E1 -27407.567,E2 -27407.567} C_VEL
LIN {X 0,Y 95.059,Z 504.886,A -85,B 0,C 180,E1 -27411.227,E2 -27411.227} C_VEL
LIN {X 0,Y 96.843,Z 542.192,A -85,B 0,C 180,E1 -27416.248,E2 -27416.248} C_VEL
LIN {X 0,Y 94.096,Z 579.194,A -85,B 0,C 180,E1 -27421.111,E2 -27421.111} C_VEL
